KUKA KRL program: ConfGarra.src, ConfGarra.dat

--- ConfGarra.src ---
&ACCESS RVO1
&PARAM EDITMASK = *
DEF ConfGarra( )

      SWITCH ConfGarraOp
         CASE 11
            Abre_Gar_Triplo_Lado_A = TRUE
            Fecha_Gar_Triplo_Lado_A = FALSE

            Abre_Gar_Triplo_Lado_B = FALSE
            Fecha_Gar_Triplo_Lado_B = TRUE

            Abre_Comp_Indiv_Gar_1 = FALSE
            Fecha_Comp_Indiv_Gar_1 = TRUE

            Abre_Comp_Indiv_Gar_3 = TRUE
            Fecha_Comp_Indiv_Gar_3 = FALSE

            Abre_Comp_Indiv_Gar_4 = FALSE
            Fecha_Comp_Indiv_Gar_4 = TRUE

            Abre_Comp_Indiv_Gar_6 = TRUE
            Fecha_Comp_Indiv_Gar_6 = FALSE

            Ava_Cil_2_Gar_1 = TRUE
            Rec_Cil_2_Gar_1 = FALSE

            Ava_Cil_2_Gar_2 = TRUE
            Rec_Cil_2_Gar_2 = FALSE

            Ava_Cil_2_Gar_3 = TRUE
            Rec_Cil_2_Gar_3 = FALSE

            Ava_Cil_2_Gar_4 = TRUE
            Rec_Cil_2_Gar_4 = FALSE

            Ava_Cil_2_Gar_5 = TRUE
            Rec_Cil_2_Gar_5 = FALSE

            Ava_Cil_2_Gar_6 = TRUE
            Rec_Cil_2_Gar_6 = FALSE

            Ava_Cil_1_Gar_1 = TRUE
            Rec_Cil_1_Gar_1 = FALSE

            Ava_Cil_1_Gar_2 = TRUE
            Rec_Cil_1_Gar_2 = FALSE

            Ava_Cil_1_Gar_3 = TRUE
            Rec_Cil_1_Gar_3 = FALSE

            Ava_Cil_1_Gar_4 = TRUE
            Rec_Cil_1_Gar_4 = FALSE

            Ava_Cil_1_Gar_5 = TRUE
            Rec_Cil_1_Gar_5 = FALSE

            Ava_Cil_1_Gar_6 = TRUE
            Rec_Cil_1_Gar_6 = FALSE

            WAIT FOR ( Cil_Comp_Triplo_A_Ava == FALSE )
            WAIT FOR ( Cil_Comp_Triplo_A_Rec == TRUE )
            WAIT FOR ( Cil_Comp_Triplo_B_Ava == TRUE )
            WAIT FOR ( Cil_Comp_Triplo_B_Rec == FALSE )
            WAIT FOR ( Cil_Comp_Indiv_Gr_1_Aber == FALSE )
            WAIT FOR ( Cil_Comp_Indiv_Gr_1_Fech == TRUE )
            WAIT FOR ( Cil_Comp_Indiv_Gr_3_Aber == TRUE )
            WAIT FOR ( Cil_Comp_Indiv_Gr_3_Fech == FALSE )
            WAIT FOR ( Cil_Comp_Indiv_Gr_4_Aber == FALSE )
            WAIT FOR ( Cil_Comp_Indiv_Gr_4_Fech == TRUE )
            WAIT FOR ( Cil_Comp_Indiv_Gr_6_Aber == TRUE )
            WAIT FOR ( Cil_Comp_Indiv_Gr_6_Fech == FALSE )
            WAIT FOR ( Cil_2_Gar_1_Ava == TRUE )
            WAIT FOR ( Cil_2_Gar_2_Ava == TRUE )
            WAIT FOR ( Cil_2_Gar_3_Ava == TRUE )
            WAIT FOR ( Cil_2_Gar_4_Ava == TRUE )
            WAIT FOR ( Cil_2_Gar_5_Ava == TRUE )
            WAIT FOR ( Cil_2_Gar_6_Ava == TRUE )
            WAIT FOR ( Cil_1_Gar_1_Ava == TRUE )
            WAIT FOR ( Cil_1_Gar_2_Ava == TRUE )
            WAIT FOR ( Cil_1_Gar_3_Ava == TRUE )
            WAIT FOR ( Cil_1_Gar_4_Ava == TRUE )
            WAIT FOR ( Cil_1_Gar_5_Ava == TRUE )
            WAIT FOR ( Cil_1_Gar_6_Ava == TRUE )

         CASE 21
            Abre_Gar_Triplo_Lado_A = FALSE
            Fecha_Gar_Triplo_Lado_A = TRUE

            Abre_Gar_Triplo_Lado_B = FALSE
            Fecha_Gar_Triplo_Lado_B = TRUE

            Abre_Comp_Indiv_Gar_1 = FALSE
            Fecha_Comp_Indiv_Gar_1 = TRUE

            Abre_Comp_Indiv_Gar_3 = FALSE
            Fecha_Comp_Indiv_Gar_3 = TRUE

            Abre_Comp_Indiv_Gar_4 = FALSE
            Fecha_Comp_Indiv_Gar_4 = TRUE

            Abre_Comp_Indiv_Gar_6 = FALSE
            Fecha_Comp_Indiv_Gar_6 = TRUE

            Ava_Cil_2_Gar_1 = TRUE
            Rec_Cil_2_Gar_1 = FALSE

            Ava_Cil_2_Gar_2 = TRUE
            Rec_Cil_2_Gar_2 = FALSE

            Ava_Cil_2_Gar_3 = TRUE
            Rec_Cil_2_Gar_3 = FALSE

            Ava_Cil_2_Gar_4 = TRUE
            Rec_Cil_2_Gar_4 = FALSE

            Ava_Cil_2_Gar_5 = TRUE
            Rec_Cil_2_Gar_5 = FALSE

            Ava_Cil_2_Gar_6 = TRUE
            Rec_Cil_2_Gar_6 = FALSE

            Ava_Cil_1_Gar_1 = TRUE
            Rec_Cil_1_Gar_1 = FALSE

            Ava_Cil_1_Gar_2 = TRUE
            Rec_Cil_1_Gar_2 = FALSE

            Ava_Cil_1_Gar_3 = TRUE
            Rec_Cil_1_Gar_3 = FALSE

            Ava_Cil_1_Gar_4 = TRUE
            Rec_Cil_1_Gar_4 = FALSE

            Ava_Cil_1_Gar_5 = TRUE
            Rec_Cil_1_Gar_5 = FALSE

            Ava_Cil_1_Gar_6 = TRUE
            Rec_Cil_1_Gar_6 = FALSE

            WAIT FOR ( Cil_Comp_Triplo_A_Ava == TRUE )
            WAIT FOR ( Cil_Comp_Triplo_A_Rec == FALSE )
            WAIT FOR ( Cil_Comp_Triplo_B_Ava == TRUE )
            WAIT FOR ( Cil_Comp_Triplo_B_Rec == FALSE )
            WAIT FOR ( Cil_Comp_Indiv_Gr_1_Aber == FALSE )
            WAIT FOR ( Cil_Comp_Indiv_Gr_1_Fech == TRUE )
            WAIT FOR ( Cil_Comp_Indiv_Gr_3_Aber == FALSE )
            WAIT FOR ( Cil_Comp_Indiv_Gr_3_Fech == TRUE )
            WAIT FOR ( Cil_Comp_Indiv_Gr_4_Aber == FALSE )
            WAIT FOR ( Cil_Comp_Indiv_Gr_4_Fech == TRUE )
            WAIT FOR ( Cil_Comp_Indiv_Gr_6_Aber == FALSE )
            WAIT FOR ( Cil_Comp_Indiv_Gr_6_Fech == TRUE )
            WAIT FOR ( Cil_2_Gar_1_Ava == TRUE )
            WAIT FOR ( Cil_2_Gar_2_Ava == TRUE )
            WAIT FOR ( Cil_2_Gar_3_Ava == TRUE )
            WAIT FOR ( Cil_2_Gar_4_Ava == TRUE )
            WAIT FOR ( Cil_2_Gar_5_Ava == TRUE )
            WAIT FOR ( Cil_2_Gar_6_Ava == TRUE )
            WAIT FOR ( Cil_1_Gar_1_Ava == TRUE )
            WAIT FOR ( Cil_1_Gar_2_Ava == TRUE )
            WAIT FOR ( Cil_1_Gar_3_Ava == TRUE )
            WAIT FOR ( Cil_1_Gar_4_Ava == TRUE )
            WAIT FOR ( Cil_1_Gar_5_Ava == TRUE )
            WAIT FOR ( Cil_1_Gar_6_Ava == TRUE )

         CASE 101
            Abre_Gar_Triplo_Lado_A = TRUE
            Fecha_Gar_Triplo_Lado_A = FALSE

            Abre_Gar_Triplo_Lado_B = TRUE
            Fecha_Gar_Triplo_Lado_B = FALSE

            Abre_Comp_Indiv_Gar_1 = TRUE
            Fecha_Comp_Indiv_Gar_1 = FALSE

            Abre_Comp_Indiv_Gar_3 = FALSE
            Fecha_Comp_Indiv_Gar_3 = TRUE

            Abre_Comp_Indiv_Gar_4 = FALSE
            Fecha_Comp_Indiv_Gar_4 = TRUE

            Abre_Comp_Indiv_Gar_6 = TRUE
            Fecha_Comp_Indiv_Gar_6 = FALSE

            Ava_Cil_2_Gar_1 = TRUE
            Rec_Cil_2_Gar_1 = FALSE

            Ava_Cil_2_Gar_2 = TRUE
            Rec_Cil_2_Gar_2 = FALSE

            Ava_Cil_2_Gar_3 = TRUE
            Rec_Cil_2_Gar_3 = FALSE

            Ava_Cil_2_Gar_4 = TRUE
            Rec_Cil_2_Gar_4 = FALSE

            Ava_Cil_2_Gar_5 = TRUE
            Rec_Cil_2_Gar_5 = FALSE

            Ava_Cil_2_Gar_6 = TRUE
            Rec_Cil_2_Gar_6 = FALSE

            Ava_Cil_1_Gar_1 = TRUE
            Rec_Cil_1_Gar_1 = FALSE

            Ava_Cil_1_Gar_2 = TRUE
            Rec_Cil_1_Gar_2 = FALSE

            Ava_Cil_1_Gar_3 = TRUE
            Rec_Cil_1_Gar_3 = FALSE

            Ava_Cil_1_Gar_4 = TRUE
            Rec_Cil_1_Gar_4 = FALSE

            Ava_Cil_1_Gar_5 = TRUE
            Rec_Cil_1_Gar_5 = FALSE

            Ava_Cil_1_Gar_6 = TRUE
            Rec_Cil_1_Gar_6 = FALSE

            WAIT FOR ( Cil_Comp_Triplo_A_Ava == FALSE )
            WAIT FOR ( Cil_Comp_Triplo_A_Rec == TRUE )
            WAIT FOR ( Cil_Comp_Triplo_B_Ava == FALSE )
            WAIT FOR ( Cil_Comp_Triplo_B_Rec == TRUE )
            WAIT FOR ( Cil_Comp_Indiv_Gr_1_Aber == TRUE )
            WAIT FOR ( Cil_Comp_Indiv_Gr_1_Fech == FALSE )
            WAIT FOR ( Cil_Comp_Indiv_Gr_3_Aber == FALSE )
            WAIT FOR ( Cil_Comp_Indiv_Gr_3_Fech == TRUE )
            WAIT FOR ( Cil_Comp_Indiv_Gr_4_Aber == FALSE )
            WAIT FOR ( Cil_Comp_Indiv_Gr_4_Fech == TRUE )
            WAIT FOR ( Cil_Comp_Indiv_Gr_6_Aber == TRUE )
            WAIT FOR ( Cil_Comp_Indiv_Gr_6_Fech == FALSE )
            WAIT FOR ( Cil_2_Gar_1_Ava == TRUE )
            WAIT FOR ( Cil_2_Gar_2_Ava == TRUE )
            WAIT FOR ( Cil_2_Gar_3_Ava == TRUE )
            WAIT FOR ( Cil_2_Gar_4_Ava == TRUE )
            WAIT FOR ( Cil_2_Gar_5_Ava == TRUE )
            WAIT FOR ( Cil_2_Gar_6_Ava == TRUE )
            WAIT FOR ( Cil_1_Gar_1_Ava == TRUE )
            WAIT FOR ( Cil_1_Gar_2_Ava == TRUE )
            WAIT FOR ( Cil_1_Gar_3_Ava == TRUE )
            WAIT FOR ( Cil_1_Gar_4_Ava == TRUE )
            WAIT FOR ( Cil_1_Gar_5_Ava == TRUE )
            WAIT FOR ( Cil_1_Gar_6_Ava == TRUE )

         CASE 102
            Abre_Gar_Triplo_Lado_A = TRUE
            Fecha_Gar_Triplo_Lado_A = FALSE

            Abre_Gar_Triplo_Lado_B = TRUE
            Fecha_Gar_Triplo_Lado_B = FALSE

            Abre_Comp_Indiv_Gar_1 = TRUE
            Fecha_Comp_Indiv_Gar_1 = FALSE

            Abre_Comp_Indiv_Gar_3 = FALSE
            Fecha_Comp_Indiv_Gar_3 = TRUE

            Abre_Comp_Indiv_Gar_4 = FALSE
            Fecha_Comp_Indiv_Gar_4 = TRUE

            Abre_Comp_Indiv_Gar_6 = TRUE
            Fecha_Comp_Indiv_Gar_6 = FALSE

            Ava_Cil_1_Gar_1 = TRUE
            Rec_Cil_1_Gar_1 = FALSE

            Ava_Cil_1_Gar_2 = TRUE
            Rec_Cil_1_Gar_2 = FALSE

            Ava_Cil_1_Gar_3 = TRUE
            Rec_Cil_1_Gar_3 = FALSE

            Ava_Cil_1_Gar_4 = TRUE
            Rec_Cil_1_Gar_4 = FALSE

            Ava_Cil_1_Gar_5 = TRUE
            Rec_Cil_1_Gar_5 = FALSE

            Ava_Cil_1_Gar_6 = TRUE
            Rec_Cil_1_Gar_6 = FALSE

            Ava_Cil_2_Gar_1 = TRUE
            Rec_Cil_2_Gar_1 = FALSE

            Ava_Cil_2_Gar_2 = TRUE
            Rec_Cil_2_Gar_2 = FALSE

            Ava_Cil_2_Gar_3 = TRUE
            Rec_Cil_2_Gar_3 = FALSE

            Ava_Cil_2_Gar_4 = TRUE
            Rec_Cil_2_Gar_4 = FALSE

            Ava_Cil_2_Gar_5 = TRUE
            Rec_Cil_2_Gar_5 = FALSE

            Ava_Cil_2_Gar_6 = TRUE
            Rec_Cil_2_Gar_6 = FALSE

            WAIT FOR ( Cil_Comp_Triplo_A_Ava == FALSE )
            WAIT FOR ( Cil_Comp_Triplo_A_Rec == TRUE )
            WAIT FOR ( Cil_Comp_Triplo_B_Ava == FALSE )
            WAIT FOR ( Cil_Comp_Triplo_B_Rec == TRUE )
            WAIT FOR ( Cil_Comp_Indiv_Gr_1_Aber == TRUE )
            WAIT FOR ( Cil_Comp_Indiv_Gr_1_Fech == FALSE )
            WAIT FOR ( Cil_Comp_Indiv_Gr_3_Aber == FALSE )
            WAIT FOR ( Cil_Comp_Indiv_Gr_3_Fech == TRUE )
            WAIT FOR ( Cil_Comp_Indiv_Gr_4_Aber == FALSE )
            WAIT FOR ( Cil_Comp_Indiv_Gr_4_Fech == TRUE )
            WAIT FOR ( Cil_Comp_Indiv_Gr_6_Aber == TRUE )
            WAIT FOR ( Cil_Comp_Indiv_Gr_6_Fech == FALSE )
            WAIT FOR ( Cil_1_Gar_1_Ava == TRUE )
            WAIT FOR ( Cil_1_Gar_2_Ava == TRUE )
            WAIT FOR ( Cil_1_Gar_3_Ava == TRUE )
            WAIT FOR ( Cil_1_Gar_4_Ava == TRUE )
            WAIT FOR ( Cil_1_Gar_5_Ava == TRUE )
            WAIT FOR ( Cil_1_Gar_6_Ava == TRUE )
            WAIT FOR ( Cil_2_Gar_1_Ava == TRUE )
            WAIT FOR ( Cil_2_Gar_2_Ava == TRUE )
            WAIT FOR ( Cil_2_Gar_3_Ava == TRUE )
            WAIT FOR ( Cil_2_Gar_4_Ava == TRUE )
            WAIT FOR ( Cil_2_Gar_5_Ava == TRUE )
            WAIT FOR ( Cil_2_Gar_6_Ava == TRUE )

         CASE 121
            Abre_Gar_Triplo_Lado_A = TRUE
            Fecha_Gar_Triplo_Lado_A = FALSE

            Abre_Gar_Triplo_Lado_B = TRUE
            Fecha_Gar_Triplo_Lado_B = FALSE

            Abre_Comp_Indiv_Gar_1 = FALSE
            Fecha_Comp_Indiv_Gar_1 = TRUE

            Abre_Comp_Indiv_Gar_3 = FALSE
            Fecha_Comp_Indiv_Gar_3 = TRUE

            Abre_Comp_Indiv_Gar_4 = FALSE
            Fecha_Comp_Indiv_Gar_4 = TRUE

            Abre_Comp_Indiv_Gar_6 = FALSE
            Fecha_Comp_Indiv_Gar_6 = TRUE

            Ava_Cil_1_Gar_1 = TRUE
            Rec_Cil_1_Gar_1 = FALSE

            Ava_Cil_1_Gar_2 = TRUE
            Rec_Cil_1_Gar_2 = FALSE

            Ava_Cil_1_Gar_3 = TRUE
            Rec_Cil_1_Gar_3 = FALSE

            Ava_Cil_1_Gar_4 = TRUE
            Rec_Cil_1_Gar_4 = FALSE

            Ava_Cil_1_Gar_5 = TRUE
            Rec_Cil_1_Gar_5 = FALSE

            Ava_Cil_1_Gar_6 = TRUE
            Rec_Cil_1_Gar_6 = FALSE

            Ava_Cil_2_Gar_1 = TRUE
            Rec_Cil_2_Gar_1 = FALSE

            Ava_Cil_2_Gar_2 = TRUE
            Rec_Cil_2_Gar_2 = FALSE

            Ava_Cil_2_Gar_3 = TRUE
            Rec_Cil_2_Gar_3 = FALSE

            Ava_Cil_2_Gar_4 = TRUE
            Rec_Cil_2_Gar_4 = FALSE

            Ava_Cil_2_Gar_5 = TRUE
            Rec_Cil_2_Gar_5 = FALSE

            Ava_Cil_2_Gar_6 = TRUE
            Rec_Cil_2_Gar_6 = FALSE

            WAIT FOR ( Cil_Comp_Triplo_A_Ava == TRUE )
            WAIT FOR ( Cil_Comp_Triplo_A_Rec == FALSE )
            WAIT FOR ( Cil_Comp_Triplo_B_Ava == TRUE )
            WAIT FOR ( Cil_Comp_Triplo_B_Rec == FALSE )
            WAIT FOR ( Cil_Comp_Indiv_Gr_1_Aber == FALSE )
            WAIT FOR ( Cil_Comp_Indiv_Gr_1_Fech == TRUE )
            WAIT FOR ( Cil_Comp_Indiv_Gr_3_Aber == FALSE )
            WAIT FOR ( Cil_Comp_Indiv_Gr_3_Fech == TRUE )
            WAIT FOR ( Cil_Comp_Indiv_Gr_4_Aber == FALSE )
            WAIT FOR ( Cil_Comp_Indiv_Gr_4_Fech == TRUE )
            WAIT FOR ( Cil_Comp_Indiv_Gr_6_Aber == FALSE )
            WAIT FOR ( Cil_Comp_Indiv_Gr_6_Fech == TRUE )
            WAIT FOR ( Cil_1_Gar_1_Ava == TRUE )
            WAIT FOR ( Cil_1_Gar_2_Ava == TRUE )
            WAIT FOR ( Cil_1_Gar_3_Ava == TRUE )
            WAIT FOR ( Cil_1_Gar_4_Ava == TRUE )
            WAIT FOR ( Cil_1_Gar_5_Ava == TRUE )
            WAIT FOR ( Cil_1_Gar_6_Ava == TRUE )
            WAIT FOR ( Cil_2_Gar_1_Ava == TRUE )
            WAIT FOR ( Cil_2_Gar_2_Ava == TRUE )
            WAIT FOR ( Cil_2_Gar_3_Ava == TRUE )
            WAIT FOR ( Cil_2_Gar_4_Ava == TRUE )
            WAIT FOR ( Cil_2_Gar_5_Ava == TRUE )
            WAIT FOR ( Cil_2_Gar_6_Ava == TRUE )

         CASE 122
            Abre_Gar_Triplo_Lado_A = TRUE
            Fecha_Gar_Triplo_Lado_A = FALSE

            Abre_Gar_Triplo_Lado_B = TRUE
            Fecha_Gar_Triplo_Lado_B = FALSE

            Abre_Comp_Indiv_Gar_1 = TRUE
            Fecha_Comp_Indiv_Gar_1 = FALSE

            Abre_Comp_Indiv_Gar_3 = FALSE
            Fecha_Comp_Indiv_Gar_3 = TRUE

            Abre_Comp_Indiv_Gar_4 = FALSE
            Fecha_Comp_Indiv_Gar_4 = TRUE

            Abre_Comp_Indiv_Gar_6 = TRUE
            Fecha_Comp_Indiv_Gar_6 = FALSE

            Ava_Cil_1_Gar_1 = TRUE
            Rec_Cil_1_Gar_1 = FALSE

            Ava_Cil_1_Gar_2 = TRUE
            Rec_Cil_1_Gar_2 = FALSE

            Ava_Cil_1_Gar_3 = TRUE
            Rec_Cil_1_Gar_3 = FALSE

            Ava_Cil_1_Gar_4 = TRUE
            Rec_Cil_1_Gar_4 = FALSE

            Ava_Cil_1_Gar_5 = TRUE
            Rec_Cil_1_Gar_5 = FALSE

            Ava_Cil_1_Gar_6 = TRUE
            Rec_Cil_1_Gar_6 = FALSE

            Ava_Cil_2_Gar_1 = TRUE
            Rec_Cil_2_Gar_1 = FALSE

            Ava_Cil_2_Gar_2 = TRUE
            Rec_Cil_2_Gar_2 = FALSE

            Ava_Cil_2_Gar_3 = TRUE
            Rec_Cil_2_Gar_3 = FALSE

            Ava_Cil_2_Gar_4 = TRUE
            Rec_Cil_2_Gar_4 = FALSE

            Ava_Cil_2_Gar_5 = TRUE
            Rec_Cil_2_Gar_5 = FALSE

            Ava_Cil_2_Gar_6 = TRUE
            Rec_Cil_2_Gar_6 = FALSE

            WAIT FOR ( Cil_Comp_Triplo_A_Ava == TRUE )
            WAIT FOR ( Cil_Comp_Triplo_A_Rec == FALSE )
            WAIT FOR ( Cil_Comp_Triplo_B_Ava == TRUE )
            WAIT FOR ( Cil_Comp_Triplo_B_Rec == FALSE )
            WAIT FOR ( Cil_Comp_Indiv_Gr_1_Aber == TRUE )
            WAIT FOR ( Cil_Comp_Indiv_Gr_1_Fech == FALSE )
            WAIT FOR ( Cil_Comp_Indiv_Gr_3_Aber == FALSE )
            WAIT FOR ( Cil_Comp_Indiv_Gr_3_Fech == TRUE )
            WAIT FOR ( Cil_Comp_Indiv_Gr_4_Aber == FALSE )
            WAIT FOR ( Cil_Comp_Indiv_Gr_4_Fech == TRUE )
            WAIT FOR ( Cil_Comp_Indiv_Gr_6_Aber == TRUE )
            WAIT FOR ( Cil_Comp_Indiv_Gr_6_Fech == FALSE )
            WAIT FOR ( Cil_1_Gar_1_Ava == TRUE )
            WAIT FOR ( Cil_1_Gar_2_Ava == TRUE )
            WAIT FOR ( Cil_1_Gar_3_Ava == TRUE )
            WAIT FOR ( Cil_1_Gar_4_Ava == TRUE )
            WAIT FOR ( Cil_1_Gar_5_Ava == TRUE )
            WAIT FOR ( Cil_1_Gar_6_Ava == TRUE )
            WAIT FOR ( Cil_2_Gar_1_Ava == TRUE )
            WAIT FOR ( Cil_2_Gar_2_Ava == TRUE )
            WAIT FOR ( Cil_2_Gar_3_Ava == TRUE )
            WAIT FOR ( Cil_2_Gar_4_Ava == TRUE )
            WAIT FOR ( Cil_2_Gar_5_Ava == TRUE )
            WAIT FOR ( Cil_2_Gar_6_Ava == TRUE )

         CASE 31
            Abre_Gar_Triplo_Lado_A = TRUE
            Fecha_Gar_Triplo_Lado_A = FALSE

            Abre_Gar_Triplo_Lado_B = TRUE
            Fecha_Gar_Triplo_Lado_B = FALSE

            Abre_Comp_Indiv_Gar_1 = FALSE
            Fecha_Comp_Indiv_Gar_1 = TRUE

            Abre_Comp_Indiv_Gar_3 = FALSE
            Fecha_Comp_Indiv_Gar_3 = TRUE

            Abre_Comp_Indiv_Gar_4 = FALSE
            Fecha_Comp_Indiv_Gar_4 = TRUE

            Abre_Comp_Indiv_Gar_6 = FALSE
            Fecha_Comp_Indiv_Gar_6 = TRUE

            Ava_Cil_1_Gar_1 = TRUE
            Rec_Cil_1_Gar_1 = FALSE

            Ava_Cil_1_Gar_2 = TRUE
            Rec_Cil_1_Gar_2 = FALSE

            Ava_Cil_1_Gar_3 = TRUE
            Rec_Cil_1_Gar_3 = FALSE

            Ava_Cil_1_Gar_4 = TRUE
            Rec_Cil_1_Gar_4 = FALSE

            Ava_Cil_1_Gar_5 = TRUE
            Rec_Cil_1_Gar_5 = FALSE

            Ava_Cil_1_Gar_6 = TRUE
            Rec_Cil_1_Gar_6 = FALSE

            Ava_Cil_2_Gar_1 = TRUE
            Rec_Cil_2_Gar_1 = FALSE

            Ava_Cil_2_Gar_2 = TRUE
            Rec_Cil_2_Gar_2 = FALSE

            Ava_Cil_2_Gar_3 = TRUE
            Rec_Cil_2_Gar_3 = FALSE

            Ava_Cil_2_Gar_4 = TRUE
            Rec_Cil_2_Gar_4 = FALSE

            Ava_Cil_2_Gar_5 = TRUE
            Rec_Cil_2_Gar_5 = FALSE

            Ava_Cil_2_Gar_6 = TRUE
            Rec_Cil_2_Gar_6 = FALSE

            WAIT FOR ( Cil_Comp_Triplo_A_Ava == TRUE )
            WAIT FOR ( Cil_Comp_Triplo_A_Rec == FALSE )
            WAIT FOR ( Cil_Comp_Triplo_B_Ava == TRUE )
            WAIT FOR ( Cil_Comp_Triplo_B_Rec == FALSE )
            WAIT FOR ( Cil_Comp_Indiv_Gr_1_Aber == FALSE )
            WAIT FOR ( Cil_Comp_Indiv_Gr_1_Fech == TRUE )
            WAIT FOR ( Cil_Comp_Indiv_Gr_3_Aber == FALSE )
            WAIT FOR ( Cil_Comp_Indiv_Gr_3_Fech == TRUE )
            WAIT FOR ( Cil_Comp_Indiv_Gr_4_Aber == FALSE )
            WAIT FOR ( Cil_Comp_Indiv_Gr_4_Fech == TRUE )
            WAIT FOR ( Cil_Comp_Indiv_Gr_6_Aber == FALSE )
            WAIT FOR ( Cil_Comp_Indiv_Gr_6_Fech == TRUE )
            WAIT FOR ( Cil_1_Gar_1_Ava == TRUE )
            WAIT FOR ( Cil_1_Gar_2_Ava == TRUE )
            WAIT FOR ( Cil_1_Gar_3_Ava == TRUE )
            WAIT FOR ( Cil_1_Gar_4_Ava == TRUE )
            WAIT FOR ( Cil_1_Gar_5_Ava == TRUE )
            WAIT FOR ( Cil_1_Gar_6_Ava == TRUE )
            WAIT FOR ( Cil_2_Gar_1_Ava == TRUE )
            WAIT FOR ( Cil_2_Gar_2_Ava == TRUE )
            WAIT FOR ( Cil_2_Gar_3_Ava == TRUE )
            WAIT FOR ( Cil_2_Gar_4_Ava == TRUE )
            WAIT FOR ( Cil_2_Gar_5_Ava == TRUE )
            WAIT FOR ( Cil_2_Gar_6_Ava == TRUE )

         CASE 32
            Abre_Gar_Triplo_Lado_A = TRUE
            Fecha_Gar_Triplo_Lado_A = FALSE

            Abre_Gar_Triplo_Lado_B = TRUE
            Fecha_Gar_Triplo_Lado_B = FALSE

            Abre_Comp_Indiv_Gar_1 = FALSE
            Fecha_Comp_Indiv_Gar_1 = TRUE

            Abre_Comp_Indiv_Gar_3 = FALSE
            Fecha_Comp_Indiv_Gar_3 = TRUE

            Abre_Comp_Indiv_Gar_4 = FALSE
            Fecha_Comp_Indiv_Gar_4 = TRUE

            Abre_Comp_Indiv_Gar_6 = FALSE
            Fecha_Comp_Indiv_Gar_6 = TRUE

            Ava_Cil_1_Gar_1 = TRUE
            Rec_Cil_1_Gar_1 = FALSE

            Ava_Cil_1_Gar_2 = TRUE
            Rec_Cil_1_Gar_2 = FALSE

            Ava_Cil_1_Gar_3 = TRUE
            Rec_Cil_1_Gar_3 = FALSE

            Ava_Cil_1_Gar_4 = TRUE
            Rec_Cil_1_Gar_4 = FALSE

            Ava_Cil_1_Gar_5 = TRUE
            Rec_Cil_1_Gar_5 = FALSE

            Ava_Cil_1_Gar_6 = TRUE
            Rec_Cil_1_Gar_6 = FALSE

            Ava_Cil_2_Gar_1 = TRUE
            Rec_Cil_2_Gar_1 = FALSE

            Ava_Cil_2_Gar_2 = TRUE
            Rec_Cil_2_Gar_2 = FALSE

            Ava_Cil_2_Gar_3 = TRUE
            Rec_Cil_2_Gar_3 = FALSE

            Ava_Cil_2_Gar_4 = TRUE
            Rec_Cil_2_Gar_4 = FALSE

            Ava_Cil_2_Gar_5 = TRUE
            Rec_Cil_2_Gar_5 = FALSE

            Ava_Cil_2_Gar_6 = TRUE
            Rec_Cil_2_Gar_6 = FALSE

            WAIT FOR ( Cil_Comp_Triplo_A_Ava == TRUE )
            WAIT FOR ( Cil_Comp_Triplo_A_Rec == FALSE )
            WAIT FOR ( Cil_Comp_Triplo_B_Ava == TRUE )
            WAIT FOR ( Cil_Comp_Triplo_B_Rec == FALSE )
            WAIT FOR ( Cil_Comp_Indiv_Gr_1_Aber == FALSE )
            WAIT FOR ( Cil_Comp_Indiv_Gr_1_Fech == TRUE )
            WAIT FOR ( Cil_Comp_Indiv_Gr_3_Aber == FALSE )
            WAIT FOR ( Cil_Comp_Indiv_Gr_3_Fech == TRUE )
            WAIT FOR ( Cil_Comp_Indiv_Gr_4_Aber == FALSE )
            WAIT FOR ( Cil_Comp_Indiv_Gr_4_Fech == TRUE )
            WAIT FOR ( Cil_Comp_Indiv_Gr_6_Aber == FALSE )
            WAIT FOR ( Cil_Comp_Indiv_Gr_6_Fech == TRUE )
            WAIT FOR ( Cil_1_Gar_1_Ava == TRUE )
            WAIT FOR ( Cil_1_Gar_2_Ava == TRUE )
            WAIT FOR ( Cil_1_Gar_3_Ava == TRUE )
            WAIT FOR ( Cil_1_Gar_4_Ava == TRUE )
            WAIT FOR ( Cil_1_Gar_5_Ava == TRUE )
            WAIT FOR ( Cil_1_Gar_6_Ava == TRUE )
            WAIT FOR ( Cil_2_Gar_1_Ava == TRUE )
            WAIT FOR ( Cil_2_Gar_2_Ava == TRUE )
            WAIT FOR ( Cil_2_Gar_3_Ava == TRUE )
            WAIT FOR ( Cil_2_Gar_4_Ava == TRUE )
            WAIT FOR ( Cil_2_Gar_5_Ava == TRUE )
            WAIT FOR ( Cil_2_Gar_6_Ava == TRUE )

         CASE 111
            Abre_Gar_Triplo_Lado_A = TRUE
            Fecha_Gar_Triplo_Lado_A = FALSE

            Abre_Gar_Triplo_Lado_B = TRUE
            Fecha_Gar_Triplo_Lado_B = FALSE

            Abre_Comp_Indiv_Gar_1 = FALSE
            Fecha_Comp_Indiv_Gar_1 = TRUE

            Abre_Comp_Indiv_Gar_3 = FALSE
            Fecha_Comp_Indiv_Gar_3 = TRUE

            Abre_Comp_Indiv_Gar_4 = FALSE
            Fecha_Comp_Indiv_Gar_4 = TRUE

            Abre_Comp_Indiv_Gar_6 = FALSE
            Fecha_Comp_Indiv_Gar_6 = TRUE

            Ava_Cil_1_Gar_1 = TRUE
            Rec_Cil_1_Gar_1 = FALSE

            Ava_Cil_1_Gar_2 = TRUE
            Rec_Cil_1_Gar_2 = FALSE

            Ava_Cil_1_Gar_3 = TRUE
            Rec_Cil_1_Gar_3 = FALSE

            Ava_Cil_1_Gar_4 = TRUE
            Rec_Cil_1_Gar_4 = FALSE

            Ava_Cil_1_Gar_5 = TRUE
            Rec_Cil_1_Gar_5 = FALSE

            Ava_Cil_1_Gar_6 = TRUE
            Rec_Cil_1_Gar_6 = FALSE

            Ava_Cil_2_Gar_1 = TRUE
            Rec_Cil_2_Gar_1 = FALSE

            Ava_Cil_2_Gar_2 = TRUE
            Rec_Cil_2_Gar_2 = FALSE

            Ava_Cil_2_Gar_3 = TRUE
            Rec_Cil_2_Gar_3 = FALSE

            Ava_Cil_2_Gar_4 = TRUE
            Rec_Cil_2_Gar_4 = FALSE

            Ava_Cil_2_Gar_5 = TRUE
            Rec_Cil_2_Gar_5 = FALSE

            Ava_Cil_2_Gar_6 = TRUE
            Rec_Cil_2_Gar_6 = FALSE

            WAIT FOR ( Cil_Comp_Triplo_A_Ava == TRUE )
            WAIT FOR ( Cil_Comp_Triplo_A_Rec == FALSE )
            WAIT FOR ( Cil_Comp_Triplo_B_Ava == TRUE )
            WAIT FOR ( Cil_Comp_Triplo_B_Rec == FALSE )
            WAIT FOR ( Cil_Comp_Indiv_Gr_1_Aber == FALSE )
            WAIT FOR ( Cil_Comp_Indiv_Gr_1_Fech == TRUE )
            WAIT FOR ( Cil_Comp_Indiv_Gr_3_Aber == FALSE )
            WAIT FOR ( Cil_Comp_Indiv_Gr_3_Fech == TRUE )
            WAIT FOR ( Cil_Comp_Indiv_Gr_4_Aber == FALSE )
            WAIT FOR ( Cil_Comp_Indiv_Gr_4_Fech == TRUE )
            WAIT FOR ( Cil_Comp_Indiv_Gr_6_Aber == FALSE )
            WAIT FOR ( Cil_Comp_Indiv_Gr_6_Fech == TRUE )
            WAIT FOR ( Cil_1_Gar_1_Ava == TRUE )
            WAIT FOR ( Cil_1_Gar_2_Ava == TRUE )
            WAIT FOR ( Cil_1_Gar_3_Ava == TRUE )
            WAIT FOR ( Cil_1_Gar_4_Ava == TRUE )
            WAIT FOR ( Cil_1_Gar_5_Ava == TRUE )
            WAIT FOR ( Cil_1_Gar_6_Ava == TRUE )
            WAIT FOR ( Cil_2_Gar_1_Ava == TRUE )
            WAIT FOR ( Cil_2_Gar_2_Ava == TRUE )
            WAIT FOR ( Cil_2_Gar_3_Ava == TRUE )
            WAIT FOR ( Cil_2_Gar_4_Ava == TRUE )
            WAIT FOR ( Cil_2_Gar_5_Ava == TRUE )
            WAIT FOR ( Cil_2_Gar_6_Ava == TRUE )

         CASE 112
            Abre_Gar_Triplo_Lado_A = TRUE
            Fecha_Gar_Triplo_Lado_A = FALSE

            Abre_Gar_Triplo_Lado_B = TRUE
            Fecha_Gar_Triplo_Lado_B = FALSE

            Abre_Comp_Indiv_Gar_1 = FALSE
            Fecha_Comp_Indiv_Gar_1 = TRUE

            Abre_Comp_Indiv_Gar_3 = FALSE
            Fecha_Comp_Indiv_Gar_3 = TRUE

            Abre_Comp_Indiv_Gar_4 = FALSE
            Fecha_Comp_Indiv_Gar_4 = TRUE

            Abre_Comp_Indiv_Gar_6 = FALSE
            Fecha_Comp_Indiv_Gar_6 = TRUE

            Ava_Cil_1_Gar_1 = TRUE
            Rec_Cil_1_Gar_1 = FALSE

            Ava_Cil_1_Gar_2 = TRUE
            Rec_Cil_1_Gar_2 = FALSE

            Ava_Cil_1_Gar_3 = TRUE
            Rec_Cil_1_Gar_3 = FALSE

            Ava_Cil_1_Gar_4 = TRUE
            Rec_Cil_1_Gar_4 = FALSE

            Ava_Cil_1_Gar_5 = TRUE
            Rec_Cil_1_Gar_5 = FALSE

            Ava_Cil_1_Gar_6 = TRUE
            Rec_Cil_1_Gar_6 = FALSE

            Ava_Cil_2_Gar_1 = TRUE
            Rec_Cil_2_Gar_1 = FALSE

            Ava_Cil_2_Gar_2 = TRUE
            Rec_Cil_2_Gar_2 = FALSE

            Ava_Cil_2_Gar_3 = TRUE
            Rec_Cil_2_Gar_3 = FALSE

            Ava_Cil_2_Gar_4 = TRUE
            Rec_Cil_2_Gar_4 = FALSE

            Ava_Cil_2_Gar_5 = TRUE
            Rec_Cil_2_Gar_5 = FALSE

            Ava_Cil_2_Gar_6 = TRUE
            Rec_Cil_2_Gar_6 = FALSE

            WAIT FOR ( Cil_Comp_Triplo_A_Ava == TRUE )
            WAIT FOR ( Cil_Comp_Triplo_A_Rec == FALSE )
            WAIT FOR ( Cil_Comp_Triplo_B_Ava == FALSE )
            WAIT FOR ( Cil_Comp_Triplo_B_Rec == TRUE )
            WAIT FOR ( Cil_Comp_Indiv_Gr_1_Aber == FALSE )
            WAIT FOR ( Cil_Comp_Indiv_Gr_1_Fech == TRUE )
            WAIT FOR ( Cil_Comp_Indiv_Gr_3_Aber == FALSE )
            WAIT FOR ( Cil_Comp_Indiv_Gr_3_Fech == TRUE )
            WAIT FOR ( Cil_Comp_Indiv_Gr_4_Aber == FALSE )
            WAIT FOR ( Cil_Comp_Indiv_Gr_4_Fech == TRUE )
            WAIT FOR ( Cil_Comp_Indiv_Gr_6_Aber == FALSE )
            WAIT FOR ( Cil_Comp_Indiv_Gr_6_Fech == TRUE )
            WAIT FOR ( Cil_1_Gar_1_Ava == TRUE )
            WAIT FOR ( Cil_1_Gar_2_Ava == TRUE )
            WAIT FOR ( Cil_1_Gar_3_Ava == TRUE )
            WAIT FOR ( Cil_1_Gar_4_Ava == TRUE )
            WAIT FOR ( Cil_1_Gar_5_Ava == TRUE )
            WAIT FOR ( Cil_1_Gar_6_Ava == TRUE )
            WAIT FOR ( Cil_2_Gar_1_Ava == TRUE )
            WAIT FOR ( Cil_2_Gar_2_Ava == TRUE )
            WAIT FOR ( Cil_2_Gar_3_Ava == TRUE )
            WAIT FOR ( Cil_2_Gar_4_Ava == TRUE )
            WAIT FOR ( Cil_2_Gar_5_Ava == TRUE )
            WAIT FOR ( Cil_2_Gar_6_Ava == TRUE )

         CASE 161
            Abre_Gar_Triplo_Lado_A = TRUE
            Fecha_Gar_Triplo_Lado_A = FALSE

            Abre_Gar_Triplo_Lado_B = TRUE
            Fecha_Gar_Triplo_Lado_B = FALSE

            Abre_Comp_Indiv_Gar_1 = FALSE
            Fecha_Comp_Indiv_Gar_1 = TRUE

            Abre_Comp_Indiv_Gar_3 = FALSE
            Fecha_Comp_Indiv_Gar_3 = TRUE

            Abre_Comp_Indiv_Gar_4 = FALSE
            Fecha_Comp_Indiv_Gar_4 = TRUE

            Abre_Comp_Indiv_Gar_6 = FALSE
            Fecha_Comp_Indiv_Gar_6 = TRUE

            Ava_Cil_1_Gar_1 = TRUE
            Rec_Cil_1_Gar_1 = FALSE

            Ava_Cil_1_Gar_2 = TRUE
            Rec_Cil_1_Gar_2 = FALSE

            Ava_Cil_1_Gar_3 = TRUE
            Rec_Cil_1_Gar_3 = FALSE

            Ava_Cil_1_Gar_4 = TRUE
            Rec_Cil_1_Gar_4 = FALSE

            Ava_Cil_1_Gar_5 = TRUE
            Rec_Cil_1_Gar_5 = FALSE

            Ava_Cil_1_Gar_6 = TRUE
            Rec_Cil_1_Gar_6 = FALSE

            Ava_Cil_2_Gar_1 = TRUE
            Rec_Cil_2_Gar_1 = FALSE

            Ava_Cil_2_Gar_2 = TRUE
            Rec_Cil_2_Gar_2 = FALSE

            Ava_Cil_2_Gar_3 = TRUE
            Rec_Cil_2_Gar_3 = FALSE

            Ava_Cil_2_Gar_4 = TRUE
            Rec_Cil_2_Gar_4 = FALSE

            Ava_Cil_2_Gar_5 = TRUE
            Rec_Cil_2_Gar_5 = FALSE

            Ava_Cil_2_Gar_6 = TRUE
            Rec_Cil_2_Gar_6 = FALSE

            WAIT FOR ( Cil_Comp_Triplo_A_Ava == TRUE )
            WAIT FOR ( Cil_Comp_Triplo_A_Rec == FALSE )
            WAIT FOR ( Cil_Comp_Triplo_B_Ava == FALSE )
            WAIT FOR ( Cil_Comp_Triplo_B_Rec == TRUE )
            WAIT FOR ( Cil_Comp_Indiv_Gr_1_Aber == FALSE )
            WAIT FOR ( Cil_Comp_Indiv_Gr_1_Fech == TRUE )
            WAIT FOR ( Cil_Comp_Indiv_Gr_3_Aber == FALSE )
            WAIT FOR ( Cil_Comp_Indiv_Gr_3_Fech == TRUE )
            WAIT FOR ( Cil_Comp_Indiv_Gr_4_Aber == FALSE )
            WAIT FOR ( Cil_Comp_Indiv_Gr_4_Fech == TRUE )
            WAIT FOR ( Cil_Comp_Indiv_Gr_6_Aber == FALSE )
            WAIT FOR ( Cil_Comp_Indiv_Gr_6_Fech == TRUE )
            WAIT FOR ( Cil_1_Gar_1_Ava == TRUE )
            WAIT FOR ( Cil_1_Gar_2_Ava == TRUE )
            WAIT FOR ( Cil_1_Gar_3_Ava == TRUE )
            WAIT FOR ( Cil_1_Gar_4_Ava == TRUE )
            WAIT FOR ( Cil_1_Gar_5_Ava == TRUE )
            WAIT FOR ( Cil_1_Gar_6_Ava == TRUE )
            WAIT FOR ( Cil_2_Gar_1_Ava == TRUE )
            WAIT FOR ( Cil_2_Gar_2_Ava == TRUE )
            WAIT FOR ( Cil_2_Gar_3_Ava == TRUE )
            WAIT FOR ( Cil_2_Gar_4_Ava == TRUE )
            WAIT FOR ( Cil_2_Gar_5_Ava == TRUE )
            WAIT FOR ( Cil_2_Gar_6_Ava == TRUE )

         CASE 162
            Abre_Gar_Triplo_Lado_A = TRUE
            Fecha_Gar_Triplo_Lado_A = FALSE

            Abre_Gar_Triplo_Lado_B = TRUE
            Fecha_Gar_Triplo_Lado_B = FALSE

            Abre_Comp_Indiv_Gar_1 = FALSE
            Fecha_Comp_Indiv_Gar_1 = TRUE

            Abre_Comp_Indiv_Gar_3 = FALSE
            Fecha_Comp_Indiv_Gar_3 = TRUE

            Abre_Comp_Indiv_Gar_4 = FALSE
            Fecha_Comp_Indiv_Gar_4 = TRUE

            Abre_Comp_Indiv_Gar_6 = TRUE
            Fecha_Comp_Indiv_Gar_6 = FALSE

            Ava_Cil_1_Gar_1 = TRUE
            Rec_Cil_1_Gar_1 = FALSE

            Ava_Cil_1_Gar_2 = TRUE
            Rec_Cil_1_Gar_2 = FALSE

            Ava_Cil_1_Gar_3 = TRUE
            Rec_Cil_1_Gar_3 = FALSE

            Ava_Cil_1_Gar_4 = TRUE
            Rec_Cil_1_Gar_4 = FALSE

            Ava_Cil_1_Gar_5 = TRUE
            Rec_Cil_1_Gar_5 = FALSE

            Ava_Cil_1_Gar_6 = TRUE
            Rec_Cil_1_Gar_6 = FALSE

            Ava_Cil_2_Gar_1 = TRUE
            Rec_Cil_2_Gar_1 = FALSE

            Ava_Cil_2_Gar_2 = TRUE
            Rec_Cil_2_Gar_2 = FALSE

            Ava_Cil_2_Gar_3 = TRUE
            Rec_Cil_2_Gar_3 = FALSE

            Ava_Cil_2_Gar_4 = TRUE
            Rec_Cil_2_Gar_4 = FALSE

            Ava_Cil_2_Gar_5 = TRUE
            Rec_Cil_2_Gar_5 = FALSE

            Ava_Cil_2_Gar_6 = TRUE
            Rec_Cil_2_Gar_6 = FALSE

            WAIT FOR ( Cil_Comp_Triplo_A_Ava == TRUE )
            WAIT FOR ( Cil_Comp_Triplo_A_Rec == FALSE )
            WAIT FOR ( Cil_Comp_Triplo_B_Ava == TRUE )
            WAIT FOR ( Cil_Comp_Triplo_B_Rec == FALSE )
            WAIT FOR ( Cil_Comp_Indiv_Gr_1_Aber == FALSE )
            WAIT FOR ( Cil_Comp_Indiv_Gr_1_Fech == TRUE )
            WAIT FOR ( Cil_Comp_Indiv_Gr_3_Aber == FALSE )
            WAIT FOR ( Cil_Comp_Indiv_Gr_3_Fech == TRUE )
            WAIT FOR ( Cil_Comp_Indiv_Gr_4_Aber == FALSE )
            WAIT FOR ( Cil_Comp_Indiv_Gr_4_Fech == TRUE )
            WAIT FOR ( Cil_Comp_Indiv_Gr_6_Aber == TRUE )
            WAIT FOR ( Cil_Comp_Indiv_Gr_6_Fech == FALSE )
            WAIT FOR ( Cil_1_Gar_1_Ava == TRUE )
            WAIT FOR ( Cil_1_Gar_2_Ava == TRUE )
            WAIT FOR ( Cil_1_Gar_3_Ava == TRUE )
            WAIT FOR ( Cil_1_Gar_4_Ava == TRUE )
            WAIT FOR ( Cil_1_Gar_5_Ava == TRUE )
            WAIT FOR ( Cil_1_Gar_6_Ava == TRUE )
            WAIT FOR ( Cil_2_Gar_1_Ava == TRUE )
            WAIT FOR ( Cil_2_Gar_2_Ava == TRUE )
            WAIT FOR ( Cil_2_Gar_3_Ava == TRUE )
            WAIT FOR ( Cil_2_Gar_4_Ava == TRUE )
            WAIT FOR ( Cil_2_Gar_5_Ava == TRUE )
            WAIT FOR ( Cil_2_Gar_6_Ava == TRUE )

         CASE 61
            Abre_Gar_Triplo_Lado_A = TRUE
            Fecha_Gar_Triplo_Lado_A = FALSE

            Abre_Gar_Triplo_Lado_B = TRUE
            Fecha_Gar_Triplo_Lado_B = FALSE

            Abre_Comp_Indiv_Gar_1 = TRUE
            Fecha_Comp_Indiv_Gar_1 = FALSE

            Abre_Comp_Indiv_Gar_3 = FALSE
            Fecha_Comp_Indiv_Gar_3 = TRUE

            Abre_Comp_Indiv_Gar_4 = FALSE
            Fecha_Comp_Indiv_Gar_4 = TRUE

            Abre_Comp_Indiv_Gar_6 = TRUE
            Fecha_Comp_Indiv_Gar_6 = FALSE

            Ava_Cil_1_Gar_1 = TRUE
            Rec_Cil_1_Gar_1 = FALSE

            Ava_Cil_1_Gar_2 = TRUE
            Rec_Cil_1_Gar_2 = FALSE

            Ava_Cil_1_Gar_3 = TRUE
            Rec_Cil_1_Gar_3 = FALSE

            Ava_Cil_1_Gar_4 = TRUE
            Rec_Cil_1_Gar_4 = FALSE

            Ava_Cil_1_Gar_5 = TRUE
            Rec_Cil_1_Gar_5 = FALSE

            Ava_Cil_1_Gar_6 = TRUE
            Rec_Cil_1_Gar_6 = FALSE

            Ava_Cil_2_Gar_1 = TRUE
            Rec_Cil_2_Gar_1 = FALSE

            Ava_Cil_2_Gar_2 = TRUE
            Rec_Cil_2_Gar_2 = FALSE

            Ava_Cil_2_Gar_3 = TRUE
            Rec_Cil_2_Gar_3 = FALSE

            Ava_Cil_2_Gar_4 = TRUE
            Rec_Cil_2_Gar_4 = FALSE

            Ava_Cil_2_Gar_5 = TRUE
            Rec_Cil_2_Gar_5 = FALSE

            Ava_Cil_2_Gar_6 = TRUE
            Rec_Cil_2_Gar_6 = FALSE

            WAIT FOR ( Cil_Comp_Triplo_A_Ava == TRUE )
            WAIT FOR ( Cil_Comp_Triplo_A_Rec == FALSE )
            WAIT FOR ( Cil_Comp_Triplo_B_Ava == TRUE )
            WAIT FOR ( Cil_Comp_Triplo_B_Rec == FALSE )
            WAIT FOR ( Cil_Comp_Indiv_Gr_1_Aber == TRUE )
            WAIT FOR ( Cil_Comp_Indiv_Gr_1_Fech == FALSE )
            WAIT FOR ( Cil_Comp_Indiv_Gr_3_Aber == FALSE )
            WAIT FOR ( Cil_Comp_Indiv_Gr_3_Fech == TRUE )
            WAIT FOR ( Cil_Comp_Indiv_Gr_4_Aber == FALSE )
            WAIT FOR ( Cil_Comp_Indiv_Gr_4_Fech == TRUE )
            WAIT FOR ( Cil_Comp_Indiv_Gr_6_Aber == TRUE )
            WAIT FOR ( Cil_Comp_Indiv_Gr_6_Fech == FALSE )
            WAIT FOR ( Cil_1_Gar_1_Ava == TRUE )
            WAIT FOR ( Cil_1_Gar_2_Ava == TRUE )
            WAIT FOR ( Cil_1_Gar_3_Ava == TRUE )
            WAIT FOR ( Cil_1_Gar_4_Ava == TRUE )
            WAIT FOR ( Cil_1_Gar_5_Ava == TRUE )
            WAIT FOR ( Cil_1_Gar_6_Ava == TRUE )
            WAIT FOR ( Cil_2_Gar_1_Ava == TRUE )
            WAIT FOR ( Cil_2_Gar_2_Ava == TRUE )
            WAIT FOR ( Cil_2_Gar_3_Ava == TRUE )
            WAIT FOR ( Cil_2_Gar_4_Ava == TRUE )
            WAIT FOR ( Cil_2_Gar_5_Ava == TRUE )
            WAIT FOR ( Cil_2_Gar_6_Ava == TRUE )

         CASE 62
            Abre_Gar_Triplo_Lado_A = TRUE
            Fecha_Gar_Triplo_Lado_A = FALSE

            Abre_Gar_Triplo_Lado_B = TRUE
            Fecha_Gar_Triplo_Lado_B = FALSE

            Abre_Comp_Indiv_Gar_1 = TRUE
            Fecha_Comp_Indiv_Gar_1 = FALSE

            Abre_Comp_Indiv_Gar_3 = FALSE
            Fecha_Comp_Indiv_Gar_3 = TRUE

            Abre_Comp_Indiv_Gar_4 = FALSE
            Fecha_Comp_Indiv_Gar_4 = TRUE

            Abre_Comp_Indiv_Gar_6 = TRUE
            Fecha_Comp_Indiv_Gar_6 = FALSE

            Ava_Cil_1_Gar_1 = TRUE
            Rec_Cil_1_Gar_1 = FALSE

            Ava_Cil_1_Gar_2 = TRUE
            Rec_Cil_1_Gar_2 = FALSE

            Ava_Cil_1_Gar_3 = TRUE
            Rec_Cil_1_Gar_3 = FALSE

            Ava_Cil_1_Gar_4 = TRUE
            Rec_Cil_1_Gar_4 = FALSE

            Ava_Cil_1_Gar_5 = TRUE
            Rec_Cil_1_Gar_5 = FALSE

            Ava_Cil_1_Gar_6 = TRUE
            Rec_Cil_1_Gar_6 = FALSE

            Ava_Cil_2_Gar_1 = TRUE
            Rec_Cil_2_Gar_1 = FALSE

            Ava_Cil_2_Gar_2 = TRUE
            Rec_Cil_2_Gar_2 = FALSE

            Ava_Cil_2_Gar_3 = TRUE
            Rec_Cil_2_Gar_3 = FALSE

            Ava_Cil_2_Gar_4 = TRUE
            Rec_Cil_2_Gar_4 = FALSE

            Ava_Cil_2_Gar_5 = TRUE
            Rec_Cil_2_Gar_5 = FALSE

            Ava_Cil_2_Gar_6 = TRUE
            Rec_Cil_2_Gar_6 = FALSE

            WAIT FOR ( Cil_Comp_Triplo_A_Ava == TRUE )
            WAIT FOR ( Cil_Comp_Triplo_A_Rec == FALSE )
            WAIT FOR ( Cil_Comp_Triplo_B_Ava == TRUE )
            WAIT FOR ( Cil_Comp_Triplo_B_Rec == FALSE )
            WAIT FOR ( Cil_Comp_Indiv_Gr_1_Aber == TRUE )
            WAIT FOR ( Cil_Comp_Indiv_Gr_1_Fech == FALSE )
            WAIT FOR ( Cil_Comp_Indiv_Gr_3_Aber == FALSE )
            WAIT FOR ( Cil_Comp_Indiv_Gr_3_Fech == TRUE )
            WAIT FOR ( Cil_Comp_Indiv_Gr_4_Aber == FALSE )
            WAIT FOR ( Cil_Comp_Indiv_Gr_4_Fech == TRUE )
            WAIT FOR ( Cil_Comp_Indiv_Gr_6_Aber == TRUE )
            WAIT FOR ( Cil_Comp_Indiv_Gr_6_Fech == FALSE )
            WAIT FOR ( Cil_1_Gar_1_Ava == TRUE )
            WAIT FOR ( Cil_1_Gar_2_Ava == TRUE )
            WAIT FOR ( Cil_1_Gar_3_Ava == TRUE )
            WAIT FOR ( Cil_1_Gar_4_Ava == TRUE )
            WAIT FOR ( Cil_1_Gar_5_Ava == TRUE )
            WAIT FOR ( Cil_1_Gar_6_Ava == TRUE )
            WAIT FOR ( Cil_2_Gar_1_Ava == TRUE )
            WAIT FOR ( Cil_2_Gar_2_Ava == TRUE )
            WAIT FOR ( Cil_2_Gar_3_Ava == TRUE )
            WAIT FOR ( Cil_2_Gar_4_Ava == TRUE )
            WAIT FOR ( Cil_2_Gar_5_Ava == TRUE )
            WAIT FOR ( Cil_2_Gar_6_Ava == TRUE )

         CASE 191
            Abre_Gar_Triplo_Lado_A = TRUE
            Fecha_Gar_Triplo_Lado_A = FALSE

            Abre_Gar_Triplo_Lado_B = TRUE
            Fecha_Gar_Triplo_Lado_B = FALSE

            Abre_Comp_Indiv_Gar_1 = FALSE
            Fecha_Comp_Indiv_Gar_1 = TRUE

            Abre_Comp_Indiv_Gar_3 = FALSE
            Fecha_Comp_Indiv_Gar_3 = TRUE

            Abre_Comp_Indiv_Gar_4 = FALSE
            Fecha_Comp_Indiv_Gar_4 = TRUE

            Abre_Comp_Indiv_Gar_6 = FALSE
            Fecha_Comp_Indiv_Gar_6 = TRUE

            Ava_Cil_1_Gar_1 = TRUE
            Rec_Cil_1_Gar_1 = FALSE

            Ava_Cil_1_Gar_2 = TRUE
            Rec_Cil_1_Gar_2 = FALSE

            Ava_Cil_1_Gar_3 = TRUE
            Rec_Cil_1_Gar_3 = FALSE

            Ava_Cil_1_Gar_4 = TRUE
            Rec_Cil_1_Gar_4 = FALSE

            Ava_Cil_1_Gar_5 = TRUE
            Rec_Cil_1_Gar_5 = FALSE

            Ava_Cil_1_Gar_6 = TRUE
            Rec_Cil_1_Gar_6 = FALSE

            Ava_Cil_2_Gar_1 = TRUE
            Rec_Cil_2_Gar_1 = FALSE

            Ava_Cil_2_Gar_2 = TRUE
            Rec_Cil_2_Gar_2 = FALSE

            Ava_Cil_2_Gar_3 = TRUE
            Rec_Cil_2_Gar_3 = FALSE

            Ava_Cil_2_Gar_4 = TRUE
            Rec_Cil_2_Gar_4 = FALSE

            Ava_Cil_2_Gar_5 = TRUE
            Rec_Cil_2_Gar_5 = FALSE

            Ava_Cil_2_Gar_6 = TRUE
            Rec_Cil_2_Gar_6 = FALSE

            WAIT FOR ( Cil_Comp_Triplo_A_Ava == TRUE )
            WAIT FOR ( Cil_Comp_Triplo_A_Rec == FALSE )
            WAIT FOR ( Cil_Comp_Triplo_B_Ava == TRUE )
            WAIT FOR ( Cil_Comp_Triplo_B_Rec == FALSE )
            WAIT FOR ( Cil_Comp_Indiv_Gr_1_Aber == FALSE )
            WAIT FOR ( Cil_Comp_Indiv_Gr_1_Fech == TRUE )
            WAIT FOR ( Cil_Comp_Indiv_Gr_3_Aber == FALSE )
            WAIT FOR ( Cil_Comp_Indiv_Gr_3_Fech == TRUE )
            WAIT FOR ( Cil_Comp_Indiv_Gr_4_Aber == FALSE )
            WAIT FOR ( Cil_Comp_Indiv_Gr_4_Fech == TRUE )
            WAIT FOR ( Cil_Comp_Indiv_Gr_6_Aber == FALSE )
            WAIT FOR ( Cil_Comp_Indiv_Gr_6_Fech == TRUE )
            WAIT FOR ( Cil_1_Gar_1_Ava == TRUE )
            WAIT FOR ( Cil_1_Gar_2_Ava == TRUE )
            WAIT FOR ( Cil_1_Gar_3_Ava == TRUE )
            WAIT FOR ( Cil_1_Gar_4_Ava == TRUE )
            WAIT FOR ( Cil_1_Gar_5_Ava == TRUE )
            WAIT FOR ( Cil_1_Gar_6_Ava == TRUE )
            WAIT FOR ( Cil_2_Gar_1_Ava == TRUE )
            WAIT FOR ( Cil_2_Gar_2_Ava == TRUE )
            WAIT FOR ( Cil_2_Gar_3_Ava == TRUE )
            WAIT FOR ( Cil_2_Gar_4_Ava == TRUE )
            WAIT FOR ( Cil_2_Gar_5_Ava == TRUE )
            WAIT FOR ( Cil_2_Gar_6_Ava == TRUE )

         CASE 192
            Abre_Gar_Triplo_Lado_A = TRUE
            Fecha_Gar_Triplo_Lado_A = FALSE

            Abre_Gar_Triplo_Lado_B = TRUE
            Fecha_Gar_Triplo_Lado_B = FALSE

            Abre_Comp_Indiv_Gar_1 = FALSE
            Fecha_Comp_Indiv_Gar_1 = TRUE

            Abre_Comp_Indiv_Gar_3 = FALSE
            Fecha_Comp_Indiv_Gar_3 = TRUE

            Abre_Comp_Indiv_Gar_4 = FALSE
            Fecha_Comp_Indiv_Gar_4 = TRUE

            Abre_Comp_Indiv_Gar_6 = FALSE
            Fecha_Comp_Indiv_Gar_6 = TRUE

            Ava_Cil_1_Gar_1 = TRUE
            Rec_Cil_1_Gar_1 = FALSE

            Ava_Cil_1_Gar_2 = TRUE
            Rec_Cil_1_Gar_2 = FALSE

            Ava_Cil_1_Gar_3 = TRUE
            Rec_Cil_1_Gar_3 = FALSE

            Ava_Cil_1_Gar_4 = TRUE
            Rec_Cil_1_Gar_4 = FALSE

            Ava_Cil_1_Gar_5 = TRUE
            Rec_Cil_1_Gar_5 = FALSE

            Ava_Cil_1_Gar_6 = TRUE
            Rec_Cil_1_Gar_6 = FALSE

            Ava_Cil_2_Gar_1 = TRUE
            Rec_Cil_2_Gar_1 = FALSE

            Ava_Cil_2_Gar_2 = TRUE
            Rec_Cil_2_Gar_2 = FALSE

            Ava_Cil_2_Gar_3 = TRUE
            Rec_Cil_2_Gar_3 = FALSE

            Ava_Cil_2_Gar_4 = TRUE
            Rec_Cil_2_Gar_4 = FALSE

            Ava_Cil_2_Gar_5 = TRUE
            Rec_Cil_2_Gar_5 = FALSE

            Ava_Cil_2_Gar_6 = TRUE
            Rec_Cil_2_Gar_6 = FALSE

            WAIT FOR ( Cil_Comp_Triplo_A_Ava == TRUE )
            WAIT FOR ( Cil_Comp_Triplo_A_Rec == FALSE )
            WAIT FOR ( Cil_Comp_Triplo_B_Ava == TRUE )
            WAIT FOR ( Cil_Comp_Triplo_B_Rec == FALSE )
            WAIT FOR ( Cil_Comp_Indiv_Gr_1_Aber == FALSE )
            WAIT FOR ( Cil_Comp_Indiv_Gr_1_Fech == TRUE )
            WAIT FOR ( Cil_Comp_Indiv_Gr_3_Aber == FALSE )
            WAIT FOR ( Cil_Comp_Indiv_Gr_3_Fech == TRUE )
            WAIT FOR ( Cil_Comp_Indiv_Gr_4_Aber == FALSE )
            WAIT FOR ( Cil_Comp_Indiv_Gr_4_Fech == TRUE )
            WAIT FOR ( Cil_Comp_Indiv_Gr_6_Aber == FALSE )
            WAIT FOR ( Cil_Comp_Indiv_Gr_6_Fech == TRUE )
            WAIT FOR ( Cil_1_Gar_1_Ava == TRUE )
            WAIT FOR ( Cil_1_Gar_2_Ava == TRUE )
            WAIT FOR ( Cil_1_Gar_3_Ava == TRUE )
            WAIT FOR ( Cil_1_Gar_4_Ava == TRUE )
            WAIT FOR ( Cil_1_Gar_5_Ava == TRUE )
            WAIT FOR ( Cil_1_Gar_6_Ava == TRUE )
            WAIT FOR ( Cil_2_Gar_1_Ava == TRUE )
            WAIT FOR ( Cil_2_Gar_2_Ava == TRUE )
            WAIT FOR ( Cil_2_Gar_3_Ava == TRUE )
            WAIT FOR ( Cil_2_Gar_4_Ava == TRUE )
            WAIT FOR ( Cil_2_Gar_5_Ava == TRUE )
            WAIT FOR ( Cil_2_Gar_6_Ava == TRUE )

         CASE 81
            Abre_Gar_Triplo_Lado_A = TRUE
            Fecha_Gar_Triplo_Lado_A = FALSE

            Abre_Gar_Triplo_Lado_B = TRUE
            Fecha_Gar_Triplo_Lado_B = FALSE

            Abre_Comp_Indiv_Gar_1 = FALSE
            Fecha_Comp_Indiv_Gar_1 = TRUE

            Abre_Comp_Indiv_Gar_3 = FALSE
            Fecha_Comp_Indiv_Gar_3 = TRUE

            Abre_Comp_Indiv_Gar_4 = FALSE
            Fecha_Comp_Indiv_Gar_4 = TRUE

            Abre_Comp_Indiv_Gar_6 = TRUE
            Fecha_Comp_Indiv_Gar_6 = FALSE

            Ava_Cil_1_Gar_1 = TRUE
            Rec_Cil_1_Gar_1 = FALSE

            Ava_Cil_1_Gar_2 = TRUE
            Rec_Cil_1_Gar_2 = FALSE

            Ava_Cil_1_Gar_3 = TRUE
            Rec_Cil_1_Gar_3 = FALSE

            Ava_Cil_1_Gar_4 = TRUE
            Rec_Cil_1_Gar_4 = FALSE

            Ava_Cil_1_Gar_5 = TRUE
            Rec_Cil_1_Gar_5 = FALSE

            Ava_Cil_1_Gar_6 = TRUE
            Rec_Cil_1_Gar_6 = FALSE

            Ava_Cil_2_Gar_1 = TRUE
            Rec_Cil_2_Gar_1 = FALSE

            Ava_Cil_2_Gar_2 = TRUE
            Rec_Cil_2_Gar_2 = FALSE

            Ava_Cil_2_Gar_3 = TRUE
            Rec_Cil_2_Gar_3 = FALSE

            Ava_Cil_2_Gar_4 = TRUE
            Rec_Cil_2_Gar_4 = FALSE

            Ava_Cil_2_Gar_5 = TRUE
            Rec_Cil_2_Gar_5 = FALSE

            Ava_Cil_2_Gar_6 = TRUE
            Rec_Cil_2_Gar_6 = FALSE

            WAIT FOR ( Cil_Comp_Triplo_A_Ava == TRUE )
            WAIT FOR ( Cil_Comp_Triplo_A_Rec == FALSE )
            WAIT FOR ( Cil_Comp_Triplo_B_Ava == TRUE )
            WAIT FOR ( Cil_Comp_Triplo_B_Rec == FALSE )
            WAIT FOR ( Cil_Comp_Indiv_Gr_1_Aber == FALSE )
            WAIT FOR ( Cil_Comp_Indiv_Gr_1_Fech == TRUE )
            WAIT FOR ( Cil_Comp_Indiv_Gr_3_Aber == FALSE )
            WAIT FOR ( Cil_Comp_Indiv_Gr_3_Fech == TRUE )
            WAIT FOR ( Cil_Comp_Indiv_Gr_4_Aber == FALSE )
            WAIT FOR ( Cil_Comp_Indiv_Gr_4_Fech == TRUE )
            WAIT FOR ( Cil_Comp_Indiv_Gr_6_Aber == TRUE )
            WAIT FOR ( Cil_Comp_Indiv_Gr_6_Fech == FALSE )
            WAIT FOR ( Cil_1_Gar_1_Ava == TRUE )
            WAIT FOR ( Cil_1_Gar_2_Ava == TRUE )
            WAIT FOR ( Cil_1_Gar_3_Ava == TRUE )
            WAIT FOR ( Cil_1_Gar_4_Ava == TRUE )
            WAIT FOR ( Cil_1_Gar_5_Ava == TRUE )
            WAIT FOR ( Cil_1_Gar_6_Ava == TRUE )
            WAIT FOR ( Cil_2_Gar_1_Ava == TRUE )
            WAIT FOR ( Cil_2_Gar_2_Ava == TRUE )
            WAIT FOR ( Cil_2_Gar_3_Ava == TRUE )
            WAIT FOR ( Cil_2_Gar_4_Ava == TRUE )
            WAIT FOR ( Cil_2_Gar_5_Ava == TRUE )
            WAIT FOR ( Cil_2_Gar_6_Ava == TRUE )

         CASE 82
            Abre_Gar_Triplo_Lado_A = TRUE
            Fecha_Gar_Triplo_Lado_A = FALSE

            Abre_Gar_Triplo_Lado_B = TRUE
            Fecha_Gar_Triplo_Lado_B = FALSE

            Abre_Comp_Indiv_Gar_1 = FALSE
            Fecha_Comp_Indiv_Gar_1 = TRUE

            Abre_Comp_Indiv_Gar_3 = TRUE
            Fecha_Comp_Indiv_Gar_3 = FALSE

            Abre_Comp_Indiv_Gar_4 = TRUE
            Fecha_Comp_Indiv_Gar_4 = FALSE

            Abre_Comp_Indiv_Gar_6 = FALSE
            Fecha_Comp_Indiv_Gar_6 = TRUE

            Ava_Cil_1_Gar_1 = TRUE
            Rec_Cil_1_Gar_1 = FALSE

            Ava_Cil_1_Gar_2 = TRUE
            Rec_Cil_1_Gar_2 = FALSE

            Ava_Cil_1_Gar_3 = TRUE
            Rec_Cil_1_Gar_3 = FALSE

            Ava_Cil_1_Gar_4 = TRUE
            Rec_Cil_1_Gar_4 = FALSE

            Ava_Cil_1_Gar_5 = TRUE
            Rec_Cil_1_Gar_5 = FALSE

            Ava_Cil_1_Gar_6 = TRUE
            Rec_Cil_1_Gar_6 = FALSE

            Ava_Cil_2_Gar_1 = TRUE
            Rec_Cil_2_Gar_1 = FALSE

            Ava_Cil_2_Gar_2 = TRUE
            Rec_Cil_2_Gar_2 = FALSE

            Ava_Cil_2_Gar_3 = TRUE
            Rec_Cil_2_Gar_3 = FALSE

            Ava_Cil_2_Gar_4 = TRUE
            Rec_Cil_2_Gar_4 = FALSE

            Ava_Cil_2_Gar_5 = TRUE
            Rec_Cil_2_Gar_5 = FALSE

            Ava_Cil_2_Gar_6 = TRUE
            Rec_Cil_2_Gar_6 = FALSE

            WAIT FOR ( Cil_Comp_Triplo_A_Ava == FALSE )
            WAIT FOR ( Cil_Comp_Triplo_A_Rec == TRUE )
            WAIT FOR ( Cil_Comp_Triplo_B_Ava == FALSE )
            WAIT FOR ( Cil_Comp_Triplo_B_Rec == TRUE )
            WAIT FOR ( Cil_Comp_Indiv_Gr_1_Aber == FALSE )
            WAIT FOR ( Cil_Comp_Indiv_Gr_1_Fech == TRUE )
            WAIT FOR ( Cil_Comp_Indiv_Gr_3_Aber == TRUE )
            WAIT FOR ( Cil_Comp_Indiv_Gr_3_Fech == FALSE )
            WAIT FOR ( Cil_Comp_Indiv_Gr_4_Aber == TRUE )
            WAIT FOR ( Cil_Comp_Indiv_Gr_4_Fech == FALSE )
            WAIT FOR ( Cil_Comp_Indiv_Gr_6_Aber == FALSE )
            WAIT FOR ( Cil_Comp_Indiv_Gr_6_Fech == TRUE )
            WAIT FOR ( Cil_1_Gar_1_Ava == TRUE )
            WAIT FOR ( Cil_1_Gar_2_Ava == TRUE )
            WAIT FOR ( Cil_1_Gar_3_Ava == TRUE )
            WAIT FOR ( Cil_1_Gar_4_Ava == TRUE )
            WAIT FOR ( Cil_1_Gar_5_Ava == TRUE )
            WAIT FOR ( Cil_1_Gar_6_Ava == TRUE )
            WAIT FOR ( Cil_2_Gar_1_Ava == TRUE )
            WAIT FOR ( Cil_2_Gar_2_Ava == TRUE )
            WAIT FOR ( Cil_2_Gar_3_Ava == TRUE )
            WAIT FOR ( Cil_2_Gar_4_Ava == TRUE )
            WAIT FOR ( Cil_2_Gar_5_Ava == TRUE )
            WAIT FOR ( Cil_2_Gar_6_Ava == TRUE )

         CASE 91
            Abre_Gar_Triplo_Lado_A = TRUE
            Fecha_Gar_Triplo_Lado_A = FALSE

            Abre_Gar_Triplo_Lado_B = TRUE
            Fecha_Gar_Triplo_Lado_B = FALSE

            Abre_Comp_Indiv_Gar_1 = FALSE
            Fecha_Comp_Indiv_Gar_1 = TRUE

            Abre_Comp_Indiv_Gar_3 = TRUE
            Fecha_Comp_Indiv_Gar_3 = FALSE

            Abre_Comp_Indiv_Gar_4 = TRUE
            Fecha_Comp_Indiv_Gar_4 = FALSE

            Abre_Comp_Indiv_Gar_6 = FALSE
            Fecha_Comp_Indiv_Gar_6 = TRUE

            Ava_Cil_1_Gar_1 = TRUE
            Rec_Cil_1_Gar_1 = FALSE

            Ava_Cil_1_Gar_2 = TRUE
            Rec_Cil_1_Gar_2 = FALSE

            Ava_Cil_1_Gar_3 = TRUE
            Rec_Cil_1_Gar_3 = FALSE

            Ava_Cil_1_Gar_4 = TRUE
            Rec_Cil_1_Gar_4 = FALSE

            Ava_Cil_1_Gar_5 = TRUE
            Rec_Cil_1_Gar_5 = FALSE

            Ava_Cil_1_Gar_6 = TRUE
            Rec_Cil_1_Gar_6 = FALSE

            Ava_Cil_2_Gar_1 = TRUE
            Rec_Cil_2_Gar_1 = FALSE

            Ava_Cil_2_Gar_2 = TRUE
            Rec_Cil_2_Gar_2 = FALSE

            Ava_Cil_2_Gar_3 = TRUE
            Rec_Cil_2_Gar_3 = FALSE

            Ava_Cil_2_Gar_4 = TRUE
            Rec_Cil_2_Gar_4 = FALSE

            Ava_Cil_2_Gar_5 = TRUE
            Rec_Cil_2_Gar_5 = FALSE

            Ava_Cil_2_Gar_6 = TRUE
            Rec_Cil_2_Gar_6 = FALSE

            WAIT FOR ( Cil_Comp_Triplo_A_Ava == FALSE )
            WAIT FOR ( Cil_Comp_Triplo_A_Rec == TRUE )
            WAIT FOR ( Cil_Comp_Triplo_B_Ava == FALSE )
            WAIT FOR ( Cil_Comp_Triplo_B_Rec == TRUE )
            WAIT FOR ( Cil_Comp_Indiv_Gr_1_Aber == FALSE )
            WAIT FOR ( Cil_Comp_Indiv_Gr_1_Fech == TRUE )
            WAIT FOR ( Cil_Comp_Indiv_Gr_3_Aber == TRUE )
            WAIT FOR ( Cil_Comp_Indiv_Gr_3_Fech == FALSE )
            WAIT FOR ( Cil_Comp_Indiv_Gr_4_Aber == TRUE )
            WAIT FOR ( Cil_Comp_Indiv_Gr_4_Fech == FALSE )
            WAIT FOR ( Cil_Comp_Indiv_Gr_6_Aber == FALSE )
            WAIT FOR ( Cil_Comp_Indiv_Gr_6_Fech == TRUE )
            WAIT FOR ( Cil_1_Gar_1_Ava == TRUE )
            WAIT FOR ( Cil_1_Gar_2_Ava == TRUE )
            WAIT FOR ( Cil_1_Gar_3_Ava == TRUE )
            WAIT FOR ( Cil_1_Gar_4_Ava == TRUE )
            WAIT FOR ( Cil_1_Gar_5_Ava == TRUE )
            WAIT FOR ( Cil_1_Gar_6_Ava == TRUE )
            WAIT FOR ( Cil_2_Gar_1_Ava == TRUE )
            WAIT FOR ( Cil_2_Gar_2_Ava == TRUE )
            WAIT FOR ( Cil_2_Gar_3_Ava == TRUE )
            WAIT FOR ( Cil_2_Gar_4_Ava == TRUE )
            WAIT FOR ( Cil_2_Gar_5_Ava == TRUE )
            WAIT FOR ( Cil_2_Gar_6_Ava == TRUE )

         CASE 92
            Abre_Gar_Triplo_Lado_A = TRUE
            Fecha_Gar_Triplo_Lado_A = FALSE

            Abre_Gar_Triplo_Lado_B = TRUE
            Fecha_Gar_Triplo_Lado_B = FALSE

            Abre_Comp_Indiv_Gar_1 = FALSE
            Fecha_Comp_Indiv_Gar_1 = TRUE

            Abre_Comp_Indiv_Gar_3 = FALSE
            Fecha_Comp_Indiv_Gar_3 = TRUE

            Abre_Comp_Indiv_Gar_4 = FALSE
            Fecha_Comp_Indiv_Gar_4 = TRUE

            Abre_Comp_Indiv_Gar_6 = TRUE
            Fecha_Comp_Indiv_Gar_6 = FALSE

            Ava_Cil_1_Gar_1 = TRUE
            Rec_Cil_1_Gar_1 = FALSE

            Ava_Cil_1_Gar_2 = TRUE
            Rec_Cil_1_Gar_2 = FALSE

            Ava_Cil_1_Gar_3 = TRUE
            Rec_Cil_1_Gar_3 = FALSE

            Ava_Cil_1_Gar_4 = TRUE
            Rec_Cil_1_Gar_4 = FALSE

            Ava_Cil_1_Gar_5 = TRUE
            Rec_Cil_1_Gar_5 = FALSE

            Ava_Cil_1_Gar_6 = TRUE
            Rec_Cil_1_Gar_6 = FALSE

            Ava_Cil_2_Gar_1 = TRUE
            Rec_Cil_2_Gar_1 = FALSE

            Ava_Cil_2_Gar_2 = TRUE
            Rec_Cil_2_Gar_2 = FALSE

            Ava_Cil_2_Gar_3 = TRUE
            Rec_Cil_2_Gar_3 = FALSE

            Ava_Cil_2_Gar_4 = TRUE
            Rec_Cil_2_Gar_4 = FALSE

            Ava_Cil_2_Gar_5 = TRUE
            Rec_Cil_2_Gar_5 = FALSE

            Ava_Cil_2_Gar_6 = TRUE
            Rec_Cil_2_Gar_6 = FALSE

            WAIT FOR ( Cil_Comp_Triplo_A_Ava == TRUE )
            WAIT FOR ( Cil_Comp_Triplo_A_Rec == FALSE )
            WAIT FOR ( Cil_Comp_Triplo_B_Ava == TRUE )
            WAIT FOR ( Cil_Comp_Triplo_B_Rec == FALSE )
            WAIT FOR ( Cil_Comp_Indiv_Gr_1_Aber == FALSE )
            WAIT FOR ( Cil_Comp_Indiv_Gr_1_Fech == TRUE )
            WAIT FOR ( Cil_Comp_Indiv_Gr_3_Aber == FALSE )
            WAIT FOR ( Cil_Comp_Indiv_Gr_3_Fech == TRUE )
            WAIT FOR ( Cil_Comp_Indiv_Gr_4_Aber == FALSE )
            WAIT FOR ( Cil_Comp_Indiv_Gr_4_Fech == TRUE )
            WAIT FOR ( Cil_Comp_Indiv_Gr_6_Aber == TRUE )
            WAIT FOR ( Cil_Comp_Indiv_Gr_6_Fech == FALSE )
            WAIT FOR ( Cil_1_Gar_1_Ava == TRUE )
            WAIT FOR ( Cil_1_Gar_2_Ava == TRUE )
            WAIT FOR ( Cil_1_Gar_3_Ava == TRUE )
            WAIT FOR ( Cil_1_Gar_4_Ava == TRUE )
            WAIT FOR ( Cil_1_Gar_5_Ava == TRUE )
            WAIT FOR ( Cil_1_Gar_6_Ava == TRUE )
            WAIT FOR ( Cil_2_Gar_1_Ava == TRUE )
            WAIT FOR ( Cil_2_Gar_2_Ava == TRUE )
            WAIT FOR ( Cil_2_Gar_3_Ava == TRUE )
            WAIT FOR ( Cil_2_Gar_4_Ava == TRUE )
            WAIT FOR ( Cil_2_Gar_5_Ava == TRUE )
            WAIT FOR ( Cil_2_Gar_6_Ava == TRUE )

         CASE 151
            Abre_Gar_Triplo_Lado_A = TRUE
            Fecha_Gar_Triplo_Lado_A = FALSE

            Abre_Gar_Triplo_Lado_B = TRUE
            Fecha_Gar_Triplo_Lado_B = FALSE

            Abre_Comp_Indiv_Gar_1 = TRUE
            Fecha_Comp_Indiv_Gar_1 = FALSE

            Abre_Comp_Indiv_Gar_3 = FALSE
            Fecha_Comp_Indiv_Gar_3 = TRUE

            Abre_Comp_Indiv_Gar_4 = FALSE
            Fecha_Comp_Indiv_Gar_4 = TRUE

            Abre_Comp_Indiv_Gar_6 = TRUE
            Fecha_Comp_Indiv_Gar_6 = FALSE

            Ava_Cil_1_Gar_1 = TRUE
            Rec_Cil_1_Gar_1 = FALSE

            Ava_Cil_1_Gar_2 = TRUE
            Rec_Cil_1_Gar_2 = FALSE

            Ava_Cil_1_Gar_3 = TRUE
            Rec_Cil_1_Gar_3 = FALSE

            Ava_Cil_1_Gar_4 = TRUE
            Rec_Cil_1_Gar_4 = FALSE

            Ava_Cil_1_Gar_5 = TRUE
            Rec_Cil_1_Gar_5 = FALSE

            Ava_Cil_1_Gar_6 = TRUE
            Rec_Cil_1_Gar_6 = FALSE

            Ava_Cil_2_Gar_1 = TRUE
            Rec_Cil_2_Gar_1 = FALSE

            Ava_Cil_2_Gar_2 = TRUE
            Rec_Cil_2_Gar_2 = FALSE

            Ava_Cil_2_Gar_3 = TRUE
            Rec_Cil_2_Gar_3 = FALSE

            Ava_Cil_2_Gar_4 = TRUE
            Rec_Cil_2_Gar_4 = FALSE

            Ava_Cil_2_Gar_5 = TRUE
            Rec_Cil_2_Gar_5 = FALSE

            Ava_Cil_2_Gar_6 = TRUE
            Rec_Cil_2_Gar_6 = FALSE

            WAIT FOR ( Cil_Comp_Triplo_A_Ava == TRUE )
            WAIT FOR ( Cil_Comp_Triplo_A_Rec == FALSE )
            WAIT FOR ( Cil_Comp_Triplo_B_Ava == TRUE )
            WAIT FOR ( Cil_Comp_Triplo_B_Rec == FALSE )
            WAIT FOR ( Cil_Comp_Indiv_Gr_1_Aber == TRUE )
            WAIT FOR ( Cil_Comp_Indiv_Gr_1_Fech == FALSE )
            WAIT FOR ( Cil_Comp_Indiv_Gr_3_Aber == FALSE )
            WAIT FOR ( Cil_Comp_Indiv_Gr_3_Fech == TRUE )
            WAIT FOR ( Cil_Comp_Indiv_Gr_4_Aber == FALSE )
            WAIT FOR ( Cil_Comp_Indiv_Gr_4_Fech == TRUE )
            WAIT FOR ( Cil_Comp_Indiv_Gr_6_Aber == TRUE )
            WAIT FOR ( Cil_Comp_Indiv_Gr_6_Fech == FALSE )
            WAIT FOR ( Cil_1_Gar_1_Ava == TRUE )
            WAIT FOR ( Cil_1_Gar_2_Ava == TRUE )
            WAIT FOR ( Cil_1_Gar_3_Ava == TRUE )
            WAIT FOR ( Cil_1_Gar_4_Ava == TRUE )
            WAIT FOR ( Cil_1_Gar_5_Ava == TRUE )
            WAIT FOR ( Cil_1_Gar_6_Ava == TRUE )
            WAIT FOR ( Cil_2_Gar_1_Ava == TRUE )
            WAIT FOR ( Cil_2_Gar_2_Ava == TRUE )
            WAIT FOR ( Cil_2_Gar_3_Ava == TRUE )
            WAIT FOR ( Cil_2_Gar_4_Ava == TRUE )
            WAIT FOR ( Cil_2_Gar_5_Ava == TRUE )
            WAIT FOR ( Cil_2_Gar_6_Ava == TRUE )

         CASE 141
            Abre_Gar_Triplo_Lado_A = TRUE
            Fecha_Gar_Triplo_Lado_A = FALSE

            Abre_Gar_Triplo_Lado_B = TRUE
            Fecha_Gar_Triplo_Lado_B = FALSE

            Abre_Comp_Indiv_Gar_1 = FALSE
            Fecha_Comp_Indiv_Gar_1 = TRUE

            Abre_Comp_Indiv_Gar_3 = FALSE
            Fecha_Comp_Indiv_Gar_3 = TRUE

            Abre_Comp_Indiv_Gar_4 = FALSE
            Fecha_Comp_Indiv_Gar_4 = TRUE

            Abre_Comp_Indiv_Gar_6 = FALSE
            Fecha_Comp_Indiv_Gar_6 = TRUE

            Ava_Cil_1_Gar_1 = TRUE
            Rec_Cil_1_Gar_1 = FALSE

            Ava_Cil_1_Gar_2 = TRUE
            Rec_Cil_1_Gar_2 = FALSE

            Ava_Cil_1_Gar_3 = TRUE
            Rec_Cil_1_Gar_3 = FALSE

            Ava_Cil_1_Gar_4 = TRUE
            Rec_Cil_1_Gar_4 = FALSE

            Ava_Cil_1_Gar_5 = TRUE
            Rec_Cil_1_Gar_5 = FALSE

            Ava_Cil_1_Gar_6 = TRUE
            Rec_Cil_1_Gar_6 = FALSE

            Ava_Cil_2_Gar_1 = TRUE
            Rec_Cil_2_Gar_1 = FALSE

            Ava_Cil_2_Gar_2 = TRUE
            Rec_Cil_2_Gar_2 = FALSE

            Ava_Cil_2_Gar_3 = TRUE
            Rec_Cil_2_Gar_3 = FALSE

            Ava_Cil_2_Gar_4 = TRUE
            Rec_Cil_2_Gar_4 = FALSE

            Ava_Cil_2_Gar_5 = TRUE
            Rec_Cil_2_Gar_5 = FALSE

            Ava_Cil_2_Gar_6 = TRUE
            Rec_Cil_2_Gar_6 = FALSE

            WAIT FOR ( Cil_Comp_Triplo_A_Ava == FALSE )
            WAIT FOR ( Cil_Comp_Triplo_A_Rec == TRUE )
            WAIT FOR ( Cil_Comp_Triplo_B_Ava == FALSE )
            WAIT FOR ( Cil_Comp_Triplo_B_Rec == TRUE )
            WAIT FOR ( Cil_Comp_Indiv_Gr_1_Aber == FALSE )
            WAIT FOR ( Cil_Comp_Indiv_Gr_1_Fech == TRUE )
            WAIT FOR ( Cil_Comp_Indiv_Gr_3_Aber == FALSE )
            WAIT FOR ( Cil_Comp_Indiv_Gr_3_Fech == TRUE )
            WAIT FOR ( Cil_Comp_Indiv_Gr_4_Aber == FALSE )
            WAIT FOR ( Cil_Comp_Indiv_Gr_4_Fech == TRUE )
            WAIT FOR ( Cil_Comp_Indiv_Gr_6_Aber == FALSE )
            WAIT FOR ( Cil_Comp_Indiv_Gr_6_Fech == TRUE )
            WAIT FOR ( Cil_1_Gar_1_Ava == TRUE )
            WAIT FOR ( Cil_1_Gar_2_Ava == TRUE )
            WAIT FOR ( Cil_1_Gar_3_Ava == TRUE )
            WAIT FOR ( Cil_1_Gar_4_Ava == TRUE )
            WAIT FOR ( Cil_1_Gar_5_Ava == TRUE )
            WAIT FOR ( Cil_1_Gar_6_Ava == TRUE )
            WAIT FOR ( Cil_2_Gar_1_Ava == TRUE )
            WAIT FOR ( Cil_2_Gar_2_Ava == TRUE )
            WAIT FOR ( Cil_2_Gar_3_Ava == TRUE )
            WAIT FOR ( Cil_2_Gar_4_Ava == TRUE )
            WAIT FOR ( Cil_2_Gar_5_Ava == TRUE )
            WAIT FOR ( Cil_2_Gar_6_Ava == TRUE )

         CASE 142
            Abre_Gar_Triplo_Lado_A = TRUE
            Fecha_Gar_Triplo_Lado_A = FALSE

            Abre_Gar_Triplo_Lado_B = TRUE
            Fecha_Gar_Triplo_Lado_B = FALSE

            Abre_Comp_Indiv_Gar_1 = FALSE
            Fecha_Comp_Indiv_Gar_1 = TRUE

            Abre_Comp_Indiv_Gar_3 = FALSE
            Fecha_Comp_Indiv_Gar_3 = TRUE

            Abre_Comp_Indiv_Gar_4 = FALSE
            Fecha_Comp_Indiv_Gar_4 = TRUE

            Abre_Comp_Indiv_Gar_6 = FALSE
            Fecha_Comp_Indiv_Gar_6 = TRUE

            Ava_Cil_1_Gar_1 = TRUE
            Rec_Cil_1_Gar_1 = FALSE

            Ava_Cil_1_Gar_2 = TRUE
            Rec_Cil_1_Gar_2 = FALSE

            Ava_Cil_1_Gar_3 = TRUE
            Rec_Cil_1_Gar_3 = FALSE

            Ava_Cil_1_Gar_4 = TRUE
            Rec_Cil_1_Gar_4 = FALSE

            Ava_Cil_1_Gar_5 = TRUE
            Rec_Cil_1_Gar_5 = FALSE

            Ava_Cil_1_Gar_6 = TRUE
            Rec_Cil_1_Gar_6 = FALSE

            Ava_Cil_2_Gar_1 = TRUE
            Rec_Cil_2_Gar_1 = FALSE

            Ava_Cil_2_Gar_2 = TRUE
            Rec_Cil_2_Gar_2 = FALSE

            Ava_Cil_2_Gar_3 = TRUE
            Rec_Cil_2_Gar_3 = FALSE

            Ava_Cil_2_Gar_4 = TRUE
            Rec_Cil_2_Gar_4 = FALSE

            Ava_Cil_2_Gar_5 = TRUE
            Rec_Cil_2_Gar_5 = FALSE

            Ava_Cil_2_Gar_6 = TRUE
            Rec_Cil_2_Gar_6 = FALSE

            WAIT FOR ( Cil_Comp_Triplo_A_Ava == FALSE )
            WAIT FOR ( Cil_Comp_Triplo_A_Rec == TRUE )
            WAIT FOR ( Cil_Comp_Triplo_B_Ava == FALSE )
            WAIT FOR ( Cil_Comp_Triplo_B_Rec == TRUE )
            WAIT FOR ( Cil_Comp_Indiv_Gr_1_Aber == FALSE )
            WAIT FOR ( Cil_Comp_Indiv_Gr_1_Fech == TRUE )
            WAIT FOR ( Cil_Comp_Indiv_Gr_3_Aber == FALSE )
            WAIT FOR ( Cil_Comp_Indiv_Gr_3_Fech == TRUE )
            WAIT FOR ( Cil_Comp_Indiv_Gr_4_Aber == FALSE )
            WAIT FOR ( Cil_Comp_Indiv_Gr_4_Fech == TRUE )
            WAIT FOR ( Cil_Comp_Indiv_Gr_6_Aber == FALSE )
            WAIT FOR ( Cil_Comp_Indiv_Gr_6_Fech == TRUE )
            WAIT FOR ( Cil_1_Gar_1_Ava == TRUE )
            WAIT FOR ( Cil_1_Gar_2_Ava == TRUE )
            WAIT FOR ( Cil_1_Gar_3_Ava == TRUE )
            WAIT FOR ( Cil_1_Gar_4_Ava == TRUE )
            WAIT FOR ( Cil_1_Gar_5_Ava == TRUE )
            WAIT FOR ( Cil_1_Gar_6_Ava == TRUE )
            WAIT FOR ( Cil_2_Gar_1_Ava == TRUE )
            WAIT FOR ( Cil_2_Gar_2_Ava == TRUE )
            WAIT FOR ( Cil_2_Gar_3_Ava == TRUE )
            WAIT FOR ( Cil_2_Gar_4_Ava == TRUE )
            WAIT FOR ( Cil_2_Gar_5_Ava == TRUE )
            WAIT FOR ( Cil_2_Gar_6_Ava == TRUE )

         CASE 171
            Abre_Gar_Triplo_Lado_A = TRUE
            Fecha_Gar_Triplo_Lado_A = FALSE

            Abre_Gar_Triplo_Lado_B = TRUE
            Fecha_Gar_Triplo_Lado_B = FALSE

            Abre_Comp_Indiv_Gar_1 = TRUE
            Fecha_Comp_Indiv_Gar_1 = FALSE

            Abre_Comp_Indiv_Gar_3 = FALSE
            Fecha_Comp_Indiv_Gar_3 = TRUE

            Abre_Comp_Indiv_Gar_4 = FALSE
            Fecha_Comp_Indiv_Gar_4 = TRUE

            Abre_Comp_Indiv_Gar_6 = FALSE
            Fecha_Comp_Indiv_Gar_6 = TRUE

            Ava_Cil_1_Gar_1 = TRUE
            Rec_Cil_1_Gar_1 = FALSE

            Ava_Cil_1_Gar_2 = TRUE
            Rec_Cil_1_Gar_2 = FALSE

            Ava_Cil_1_Gar_3 = TRUE
            Rec_Cil_1_Gar_3 = FALSE

            Ava_Cil_1_Gar_4 = TRUE
            Rec_Cil_1_Gar_4 = FALSE

            Ava_Cil_1_Gar_5 = TRUE
            Rec_Cil_1_Gar_5 = FALSE

            Ava_Cil_1_Gar_6 = TRUE
            Rec_Cil_1_Gar_6 = FALSE

            Ava_Cil_2_Gar_1 = TRUE
            Rec_Cil_2_Gar_1 = FALSE

            Ava_Cil_2_Gar_2 = TRUE
            Rec_Cil_2_Gar_2 = FALSE

            Ava_Cil_2_Gar_3 = TRUE
            Rec_Cil_2_Gar_3 = FALSE

            Ava_Cil_2_Gar_4 = TRUE
            Rec_Cil_2_Gar_4 = FALSE

            Ava_Cil_2_Gar_5 = TRUE
            Rec_Cil_2_Gar_5 = FALSE

            Ava_Cil_2_Gar_6 = TRUE
            Rec_Cil_2_Gar_6 = FALSE

            WAIT FOR ( Cil_Comp_Triplo_A_Ava == TRUE )
            WAIT FOR ( Cil_Comp_Triplo_A_Rec == FALSE )
            WAIT FOR ( Cil_Comp_Triplo_B_Ava == TRUE )
            WAIT FOR ( Cil_Comp_Triplo_B_Rec == FALSE )
            WAIT FOR ( Cil_Comp_Indiv_Gr_1_Aber == TRUE )
            WAIT FOR ( Cil_Comp_Indiv_Gr_1_Fech == FALSE )
            WAIT FOR ( Cil_Comp_Indiv_Gr_3_Aber == FALSE )
            WAIT FOR ( Cil_Comp_Indiv_Gr_3_Fech == TRUE )
            WAIT FOR ( Cil_Comp_Indiv_Gr_4_Aber == FALSE )
            WAIT FOR ( Cil_Comp_Indiv_Gr_4_Fech == TRUE )
            WAIT FOR ( Cil_Comp_Indiv_Gr_6_Aber == FALSE )
            WAIT FOR ( Cil_Comp_Indiv_Gr_6_Fech == TRUE )
            WAIT FOR ( Cil_1_Gar_1_Ava == TRUE )
            WAIT FOR ( Cil_1_Gar_2_Ava == TRUE )
            WAIT FOR ( Cil_1_Gar_3_Ava == TRUE )
            WAIT FOR ( Cil_1_Gar_4_Ava == TRUE )
            WAIT FOR ( Cil_1_Gar_5_Ava == TRUE )
            WAIT FOR ( Cil_1_Gar_6_Ava == TRUE )
            WAIT FOR ( Cil_2_Gar_1_Ava == TRUE )
            WAIT FOR ( Cil_2_Gar_2_Ava == TRUE )
            WAIT FOR ( Cil_2_Gar_3_Ava == TRUE )
            WAIT FOR ( Cil_2_Gar_4_Ava == TRUE )
            WAIT FOR ( Cil_2_Gar_5_Ava == TRUE )
            WAIT FOR ( Cil_2_Gar_6_Ava == TRUE )

         CASE 172
            Abre_Gar_Triplo_Lado_A = TRUE
            Fecha_Gar_Triplo_Lado_A = FALSE

            Abre_Gar_Triplo_Lado_B = TRUE
            Fecha_Gar_Triplo_Lado_B = FALSE

            Abre_Comp_Indiv_Gar_1 = TRUE
            Fecha_Comp_Indiv_Gar_1 = FALSE

            Abre_Comp_Indiv_Gar_3 = FALSE
            Fecha_Comp_Indiv_Gar_3 = TRUE

            Abre_Comp_Indiv_Gar_4 = FALSE
            Fecha_Comp_Indiv_Gar_4 = TRUE

            Abre_Comp_Indiv_Gar_6 = TRUE
            Fecha_Comp_Indiv_Gar_6 = FALSE

            Ava_Cil_1_Gar_1 = TRUE
            Rec_Cil_1_Gar_1 = FALSE

            Ava_Cil_1_Gar_2 = TRUE
            Rec_Cil_1_Gar_2 = FALSE

            Ava_Cil_1_Gar_3 = TRUE
            Rec_Cil_1_Gar_3 = FALSE

            Ava_Cil_1_Gar_4 = TRUE
            Rec_Cil_1_Gar_4 = FALSE

            Ava_Cil_1_Gar_5 = TRUE
            Rec_Cil_1_Gar_5 = FALSE

            Ava_Cil_1_Gar_6 = TRUE
            Rec_Cil_1_Gar_6 = FALSE

            Ava_Cil_2_Gar_1 = TRUE
            Rec_Cil_2_Gar_1 = FALSE

            Ava_Cil_2_Gar_2 = TRUE
            Rec_Cil_2_Gar_2 = FALSE

            Ava_Cil_2_Gar_3 = TRUE
            Rec_Cil_2_Gar_3 = FALSE

            Ava_Cil_2_Gar_4 = TRUE
            Rec_Cil_2_Gar_4 = FALSE

            Ava_Cil_2_Gar_5 = TRUE
            Rec_Cil_2_Gar_5 = FALSE

            Ava_Cil_2_Gar_6 = TRUE
            Rec_Cil_2_Gar_6 = FALSE

            WAIT FOR ( Cil_Comp_Triplo_A_Ava == FALSE )
            WAIT FOR ( Cil_Comp_Triplo_A_Rec == TRUE )
            WAIT FOR ( Cil_Comp_Triplo_B_Ava == FALSE )
            WAIT FOR ( Cil_Comp_Triplo_B_Rec == TRUE )
            WAIT FOR ( Cil_Comp_Indiv_Gr_1_Aber == TRUE )
            WAIT FOR ( Cil_Comp_Indiv_Gr_1_Fech == FALSE )
            WAIT FOR ( Cil_Comp_Indiv_Gr_3_Aber == FALSE )
            WAIT FOR ( Cil_Comp_Indiv_Gr_3_Fech == TRUE )
            WAIT FOR ( Cil_Comp_Indiv_Gr_4_Aber == FALSE )
            WAIT FOR ( Cil_Comp_Indiv_Gr_4_Fech == TRUE )
            WAIT FOR ( Cil_Comp_Indiv_Gr_6_Aber == TRUE )
            WAIT FOR ( Cil_Comp_Indiv_Gr_6_Fech == FALSE )
            WAIT FOR ( Cil_1_Gar_1_Ava == TRUE )
            WAIT FOR ( Cil_1_Gar_2_Ava == TRUE )
            WAIT FOR ( Cil_1_Gar_3_Ava == TRUE )
            WAIT FOR ( Cil_1_Gar_4_Ava == TRUE )
            WAIT FOR ( Cil_1_Gar_5_Ava == TRUE )
            WAIT FOR ( Cil_1_Gar_6_Ava == TRUE )
            WAIT FOR ( Cil_2_Gar_1_Ava == TRUE )
            WAIT FOR ( Cil_2_Gar_2_Ava == TRUE )
            WAIT FOR ( Cil_2_Gar_3_Ava == TRUE )
            WAIT FOR ( Cil_2_Gar_4_Ava == TRUE )
            WAIT FOR ( Cil_2_Gar_5_Ava == TRUE )
            WAIT FOR ( Cil_2_Gar_6_Ava == TRUE )

         CASE 173
            Abre_Gar_Triplo_Lado_A = TRUE
            Fecha_Gar_Triplo_Lado_A = FALSE

            Abre_Gar_Triplo_Lado_B = TRUE
            Fecha_Gar_Triplo_Lado_B = FALSE

            Abre_Comp_Indiv_Gar_1 = TRUE
            Fecha_Comp_Indiv_Gar_1 = FALSE

            Abre_Comp_Indiv_Gar_3 = FALSE
            Fecha_Comp_Indiv_Gar_3 = TRUE

            Abre_Comp_Indiv_Gar_4 = FALSE
            Fecha_Comp_Indiv_Gar_4 = TRUE

            Abre_Comp_Indiv_Gar_6 = TRUE
            Fecha_Comp_Indiv_Gar_6 = FALSE

            Ava_Cil_1_Gar_1 = TRUE
            Rec_Cil_1_Gar_1 = FALSE

            Ava_Cil_1_Gar_2 = TRUE
            Rec_Cil_1_Gar_2 = FALSE

            Ava_Cil_1_Gar_3 = TRUE
            Rec_Cil_1_Gar_3 = FALSE

            Ava_Cil_1_Gar_4 = TRUE
            Rec_Cil_1_Gar_4 = FALSE

            Ava_Cil_1_Gar_5 = TRUE
            Rec_Cil_1_Gar_5 = FALSE

            Ava_Cil_1_Gar_6 = TRUE
            Rec_Cil_1_Gar_6 = FALSE

            Ava_Cil_2_Gar_1 = TRUE
            Rec_Cil_2_Gar_1 = FALSE

            Ava_Cil_2_Gar_2 = TRUE
            Rec_Cil_2_Gar_2 = FALSE

            Ava_Cil_2_Gar_3 = TRUE
            Rec_Cil_2_Gar_3 = FALSE

            Ava_Cil_2_Gar_4 = TRUE
            Rec_Cil_2_Gar_4 = FALSE

            Ava_Cil_2_Gar_5 = TRUE
            Rec_Cil_2_Gar_5 = FALSE

            Ava_Cil_2_Gar_6 = TRUE
            Rec_Cil_2_Gar_6 = FALSE

            WAIT FOR ( Cil_Comp_Triplo_A_Ava == FALSE )
            WAIT FOR ( Cil_Comp_Triplo_A_Rec == TRUE )
            WAIT FOR ( Cil_Comp_Triplo_B_Ava == FALSE )
            WAIT FOR ( Cil_Comp_Triplo_B_Rec == TRUE )
            WAIT FOR ( Cil_Comp_Indiv_Gr_1_Aber == TRUE )
            WAIT FOR ( Cil_Comp_Indiv_Gr_1_Fech == FALSE )
            WAIT FOR ( Cil_Comp_Indiv_Gr_3_Aber == FALSE )
            WAIT FOR ( Cil_Comp_Indiv_Gr_3_Fech == TRUE )
            WAIT FOR ( Cil_Comp_Indiv_Gr_4_Aber == FALSE )
            WAIT FOR ( Cil_Comp_Indiv_Gr_4_Fech == TRUE )
            WAIT FOR ( Cil_Comp_Indiv_Gr_6_Aber == TRUE )
            WAIT FOR ( Cil_Comp_Indiv_Gr_6_Fech == FALSE )
            WAIT FOR ( Cil_1_Gar_1_Ava == TRUE )
            WAIT FOR ( Cil_1_Gar_2_Ava == TRUE )
            WAIT FOR ( Cil_1_Gar_3_Ava == TRUE )
            WAIT FOR ( Cil_1_Gar_4_Ava == TRUE )
            WAIT FOR ( Cil_1_Gar_5_Ava == TRUE )
            WAIT FOR ( Cil_1_Gar_6_Ava == TRUE )
            WAIT FOR ( Cil_2_Gar_1_Ava == TRUE )
            WAIT FOR ( Cil_2_Gar_2_Ava == TRUE )
            WAIT FOR ( Cil_2_Gar_3_Ava == TRUE )
            WAIT FOR ( Cil_2_Gar_4_Ava == TRUE )
            WAIT FOR ( Cil_2_Gar_5_Ava == TRUE )
            WAIT FOR ( Cil_2_Gar_6_Ava == TRUE )

         CASE 71
            Abre_Gar_Triplo_Lado_A = TRUE
            Fecha_Gar_Triplo_Lado_A = FALSE

            Abre_Gar_Triplo_Lado_B = TRUE
            Fecha_Gar_Triplo_Lado_B = FALSE

            Abre_Comp_Indiv_Gar_1 = FALSE
            Fecha_Comp_Indiv_Gar_1 = TRUE

            Abre_Comp_Indiv_Gar_3 = TRUE
            Fecha_Comp_Indiv_Gar_3 = FALSE

            Abre_Comp_Indiv_Gar_4 = TRUE
            Fecha_Comp_Indiv_Gar_4 = FALSE

            Abre_Comp_Indiv_Gar_6 = FALSE
            Fecha_Comp_Indiv_Gar_6 = TRUE

            Ava_Cil_1_Gar_1 = TRUE
            Rec_Cil_1_Gar_1 = FALSE

            Ava_Cil_1_Gar_2 = TRUE
            Rec_Cil_1_Gar_2 = FALSE

            Ava_Cil_1_Gar_3 = TRUE
            Rec_Cil_1_Gar_3 = FALSE

            Ava_Cil_1_Gar_4 = TRUE
            Rec_Cil_1_Gar_4 = FALSE

            Ava_Cil_1_Gar_5 = TRUE
            Rec_Cil_1_Gar_5 = FALSE

            Ava_Cil_1_Gar_6 = TRUE
            Rec_Cil_1_Gar_6 = FALSE

            Ava_Cil_2_Gar_1 = TRUE
            Rec_Cil_2_Gar_1 = FALSE

            Ava_Cil_2_Gar_2 = TRUE
            Rec_Cil_2_Gar_2 = FALSE

            Ava_Cil_2_Gar_3 = TRUE
            Rec_Cil_2_Gar_3 = FALSE

            Ava_Cil_2_Gar_4 = TRUE
            Rec_Cil_2_Gar_4 = FALSE

            Ava_Cil_2_Gar_5 = TRUE
            Rec_Cil_2_Gar_5 = FALSE

            Ava_Cil_2_Gar_6 = TRUE
            Rec_Cil_2_Gar_6 = FALSE

            WAIT FOR ( Cil_Comp_Triplo_A_Ava == FALSE )
            WAIT FOR ( Cil_Comp_Triplo_A_Rec == TRUE )
            WAIT FOR ( Cil_Comp_Triplo_B_Ava == FALSE )
            WAIT FOR ( Cil_Comp_Triplo_B_Rec == TRUE )
            WAIT FOR ( Cil_Comp_Indiv_Gr_1_Aber == FALSE )
            WAIT FOR ( Cil_Comp_Indiv_Gr_1_Fech == TRUE )
            WAIT FOR ( Cil_Comp_Indiv_Gr_3_Aber == TRUE )
            WAIT FOR ( Cil_Comp_Indiv_Gr_3_Fech == FALSE )
            WAIT FOR ( Cil_Comp_Indiv_Gr_4_Aber == TRUE )
            WAIT FOR ( Cil_Comp_Indiv_Gr_4_Fech == FALSE )
            WAIT FOR ( Cil_Comp_Indiv_Gr_6_Aber == FALSE )
            WAIT FOR ( Cil_Comp_Indiv_Gr_6_Fech == TRUE )
            WAIT FOR ( Cil_1_Gar_1_Ava == TRUE )
            WAIT FOR ( Cil_1_Gar_2_Ava == TRUE )
            WAIT FOR ( Cil_1_Gar_3_Ava == TRUE )
            WAIT FOR ( Cil_1_Gar_4_Ava == TRUE )
            WAIT FOR ( Cil_1_Gar_5_Ava == TRUE )
            WAIT FOR ( Cil_1_Gar_6_Ava == TRUE )
            WAIT FOR ( Cil_2_Gar_1_Ava == TRUE )
            WAIT FOR ( Cil_2_Gar_2_Ava == TRUE )
            WAIT FOR ( Cil_2_Gar_3_Ava == TRUE )
            WAIT FOR ( Cil_2_Gar_4_Ava == TRUE )
            WAIT FOR ( Cil_2_Gar_5_Ava == TRUE )
            WAIT FOR ( Cil_2_Gar_6_Ava == TRUE )

         CASE 72
            Abre_Gar_Triplo_Lado_A = TRUE
            Fecha_Gar_Triplo_Lado_A = FALSE

            Abre_Gar_Triplo_Lado_B = TRUE
            Fecha_Gar_Triplo_Lado_B = FALSE

            Abre_Comp_Indiv_Gar_1 = TRUE
            Fecha_Comp_Indiv_Gar_1 = FALSE

            Abre_Comp_Indiv_Gar_3 = FALSE
            Fecha_Comp_Indiv_Gar_3 = TRUE

            Abre_Comp_Indiv_Gar_4 = TRUE
            Fecha_Comp_Indiv_Gar_4 = FALSE

            Abre_Comp_Indiv_Gar_6 = FALSE
            Fecha_Comp_Indiv_Gar_6 = TRUE

            Ava_Cil_1_Gar_1 = TRUE
            Rec_Cil_1_Gar_1 = FALSE

            Ava_Cil_1_Gar_2 = TRUE
            Rec_Cil_1_Gar_2 = FALSE

            Ava_Cil_1_Gar_3 = TRUE
            Rec_Cil_1_Gar_3 = FALSE

            Ava_Cil_1_Gar_4 = TRUE
            Rec_Cil_1_Gar_4 = FALSE

            Ava_Cil_1_Gar_5 = TRUE
            Rec_Cil_1_Gar_5 = FALSE

            Ava_Cil_1_Gar_6 = TRUE
            Rec_Cil_1_Gar_6 = FALSE

            Ava_Cil_2_Gar_1 = TRUE
            Rec_Cil_2_Gar_1 = FALSE

            Ava_Cil_2_Gar_2 = TRUE
            Rec_Cil_2_Gar_2 = FALSE

            Ava_Cil_2_Gar_3 = TRUE
            Rec_Cil_2_Gar_3 = FALSE

            Ava_Cil_2_Gar_4 = TRUE
            Rec_Cil_2_Gar_4 = FALSE

            Ava_Cil_2_Gar_5 = TRUE
            Rec_Cil_2_Gar_5 = FALSE

            Ava_Cil_2_Gar_6 = TRUE
            Rec_Cil_2_Gar_6 = FALSE

            WAIT FOR ( Cil_Comp_Triplo_A_Ava == FALSE )
            WAIT FOR ( Cil_Comp_Triplo_A_Rec == TRUE )
            WAIT FOR ( Cil_Comp_Triplo_B_Ava == FALSE )
            WAIT FOR ( Cil_Comp_Triplo_B_Rec == TRUE )
            WAIT FOR ( Cil_Comp_Indiv_Gr_1_Aber == TRUE )
            WAIT FOR ( Cil_Comp_Indiv_Gr_1_Fech == FALSE )
            WAIT FOR ( Cil_Comp_Indiv_Gr_3_Aber == FALSE )
            WAIT FOR ( Cil_Comp_Indiv_Gr_3_Fech == TRUE )
            WAIT FOR ( Cil_Comp_Indiv_Gr_4_Aber == TRUE )
            WAIT FOR ( Cil_Comp_Indiv_Gr_4_Fech == FALSE )
            WAIT FOR ( Cil_Comp_Indiv_Gr_6_Aber == FALSE )
            WAIT FOR ( Cil_Comp_Indiv_Gr_6_Fech == TRUE )
            WAIT FOR ( Cil_1_Gar_1_Ava == TRUE )
            WAIT FOR ( Cil_1_Gar_2_Ava == TRUE )
            WAIT FOR ( Cil_1_Gar_3_Ava == TRUE )
            WAIT FOR ( Cil_1_Gar_4_Ava == TRUE )
            WAIT FOR ( Cil_1_Gar_5_Ava == TRUE )
            WAIT FOR ( Cil_1_Gar_6_Ava == TRUE )
            WAIT FOR ( Cil_2_Gar_1_Ava == TRUE )
            WAIT FOR ( Cil_2_Gar_2_Ava == TRUE )
            WAIT FOR ( Cil_2_Gar_3_Ava == TRUE )
            WAIT FOR ( Cil_2_Gar_4_Ava == TRUE )
            WAIT FOR ( Cil_2_Gar_5_Ava == TRUE )
            WAIT FOR ( Cil_2_Gar_6_Ava == TRUE )

         CASE 73
            Abre_Gar_Triplo_Lado_A = TRUE
            Fecha_Gar_Triplo_Lado_A = FALSE

            Abre_Gar_Triplo_Lado_B = TRUE
            Fecha_Gar_Triplo_Lado_B = FALSE

            Abre_Comp_Indiv_Gar_1 = TRUE
            Fecha_Comp_Indiv_Gar_1 = FALSE

            Abre_Comp_Indiv_Gar_3 = TRUE
            Fecha_Comp_Indiv_Gar_3 = FALSE

            Abre_Comp_Indiv_Gar_4 = TRUE
            Fecha_Comp_Indiv_Gar_4 = FALSE

            Abre_Comp_Indiv_Gar_6 = TRUE
            Fecha_Comp_Indiv_Gar_6 = FALSE

            Ava_Cil_1_Gar_1 = TRUE
            Rec_Cil_1_Gar_1 = FALSE

            Ava_Cil_1_Gar_2 = TRUE
            Rec_Cil_1_Gar_2 = FALSE

            Ava_Cil_1_Gar_3 = TRUE
            Rec_Cil_1_Gar_3 = FALSE

            Ava_Cil_1_Gar_4 = TRUE
            Rec_Cil_1_Gar_4 = FALSE

            Ava_Cil_1_Gar_5 = TRUE
            Rec_Cil_1_Gar_5 = FALSE

            Ava_Cil_1_Gar_6 = TRUE
            Rec_Cil_1_Gar_6 = FALSE

            Ava_Cil_2_Gar_1 = TRUE
            Rec_Cil_2_Gar_1 = FALSE

            Ava_Cil_2_Gar_2 = TRUE
            Rec_Cil_2_Gar_2 = FALSE

            Ava_Cil_2_Gar_3 = TRUE
            Rec_Cil_2_Gar_3 = FALSE

            Ava_Cil_2_Gar_4 = TRUE
            Rec_Cil_2_Gar_4 = FALSE

            Ava_Cil_2_Gar_5 = TRUE
            Rec_Cil_2_Gar_5 = FALSE

            Ava_Cil_2_Gar_6 = TRUE
            Rec_Cil_2_Gar_6 = FALSE

            WAIT FOR ( Cil_Comp_Triplo_A_Ava == FALSE )
            WAIT FOR ( Cil_Comp_Triplo_A_Rec == TRUE )
            WAIT FOR ( Cil_Comp_Triplo_B_Ava == FALSE )
            WAIT FOR ( Cil_Comp_Triplo_B_Rec == TRUE )
            WAIT FOR ( Cil_Comp_Indiv_Gr_1_Aber == TRUE )
            WAIT FOR ( Cil_Comp_Indiv_Gr_1_Fech == FALSE )
            WAIT FOR ( Cil_Comp_Indiv_Gr_3_Aber == TRUE )
            WAIT FOR ( Cil_Comp_Indiv_Gr_3_Fech == FALSE )
            WAIT FOR ( Cil_Comp_Indiv_Gr_4_Aber == TRUE )
            WAIT FOR ( Cil_Comp_Indiv_Gr_4_Fech == FALSE )
            WAIT FOR ( Cil_Comp_Indiv_Gr_6_Aber == TRUE )
            WAIT FOR ( Cil_Comp_Indiv_Gr_6_Fech == FALSE )
            WAIT FOR ( Cil_1_Gar_1_Ava == TRUE )
            WAIT FOR ( Cil_1_Gar_2_Ava == TRUE )
            WAIT FOR ( Cil_1_Gar_3_Ava == TRUE )
            WAIT FOR ( Cil_1_Gar_4_Ava == TRUE )
            WAIT FOR ( Cil_1_Gar_5_Ava == TRUE )
            WAIT FOR ( Cil_1_Gar_6_Ava == TRUE )
            WAIT FOR ( Cil_2_Gar_1_Ava == TRUE )
            WAIT FOR ( Cil_2_Gar_2_Ava == TRUE )
            WAIT FOR ( Cil_2_Gar_3_Ava == TRUE )
            WAIT FOR ( Cil_2_Gar_4_Ava == TRUE )
            WAIT FOR ( Cil_2_Gar_5_Ava == TRUE )
            WAIT FOR ( Cil_2_Gar_6_Ava == TRUE )

         CASE 51
            Abre_Gar_Triplo_Lado_A = TRUE
            Fecha_Gar_Triplo_Lado_A = FALSE

            Abre_Gar_Triplo_Lado_B = TRUE
            Fecha_Gar_Triplo_Lado_B = FALSE

            Abre_Comp_Indiv_Gar_1 = TRUE
            Fecha_Comp_Indiv_Gar_1 = FALSE

            Abre_Comp_Indiv_Gar_3 = TRUE
            Fecha_Comp_Indiv_Gar_3 = FALSE

            Abre_Comp_Indiv_Gar_4 = TRUE
            Fecha_Comp_Indiv_Gar_4 = FALSE

            Abre_Comp_Indiv_Gar_6 = TRUE
            Fecha_Comp_Indiv_Gar_6 = FALSE

            Ava_Cil_1_Gar_1 = TRUE
            Rec_Cil_1_Gar_1 = FALSE

            Ava_Cil_1_Gar_2 = TRUE
            Rec_Cil_1_Gar_2 = FALSE

            Ava_Cil_1_Gar_3 = TRUE
            Rec_Cil_1_Gar_3 = FALSE

            Ava_Cil_1_Gar_4 = TRUE
            Rec_Cil_1_Gar_4 = FALSE

            Ava_Cil_1_Gar_5 = TRUE
            Rec_Cil_1_Gar_5 = FALSE

            Ava_Cil_1_Gar_6 = TRUE
            Rec_Cil_1_Gar_6 = FALSE

            Ava_Cil_2_Gar_1 = TRUE
            Rec_Cil_2_Gar_1 = FALSE

            Ava_Cil_2_Gar_2 = TRUE
            Rec_Cil_2_Gar_2 = FALSE

            Ava_Cil_2_Gar_3 = TRUE
            Rec_Cil_2_Gar_3 = FALSE

            Ava_Cil_2_Gar_4 = TRUE
            Rec_Cil_2_Gar_4 = FALSE

            Ava_Cil_2_Gar_5 = TRUE
            Rec_Cil_2_Gar_5 = FALSE

            Ava_Cil_2_Gar_6 = TRUE
            Rec_Cil_2_Gar_6 = FALSE

            WAIT FOR ( Cil_Comp_Triplo_A_Ava == FALSE )
            WAIT FOR ( Cil_Comp_Triplo_A_Rec == TRUE )
            WAIT FOR ( Cil_Comp_Triplo_B_Ava == FALSE )
            WAIT FOR ( Cil_Comp_Triplo_B_Rec == TRUE )
            WAIT FOR ( Cil_Comp_Indiv_Gr_1_Aber == TRUE )
            WAIT FOR ( Cil_Comp_Indiv_Gr_1_Fech == FALSE )
            WAIT FOR ( Cil_Comp_Indiv_Gr_3_Aber == TRUE )
            WAIT FOR ( Cil_Comp_Indiv_Gr_3_Fech == FALSE )
            WAIT FOR ( Cil_Comp_Indiv_Gr_4_Aber == TRUE )
            WAIT FOR ( Cil_Comp_Indiv_Gr_4_Fech == FALSE )
            WAIT FOR ( Cil_Comp_Indiv_Gr_6_Aber == TRUE )
            WAIT FOR ( Cil_Comp_Indiv_Gr_6_Fech == FALSE )
            WAIT FOR ( Cil_1_Gar_1_Ava == TRUE )
            WAIT FOR ( Cil_1_Gar_2_Ava == TRUE )
            WAIT FOR ( Cil_1_Gar_3_Ava == TRUE )
            WAIT FOR ( Cil_1_Gar_4_Ava == TRUE )
            WAIT FOR ( Cil_1_Gar_5_Ava == TRUE )
            WAIT FOR ( Cil_1_Gar_6_Ava == TRUE )
            WAIT FOR ( Cil_2_Gar_1_Ava == TRUE )
            WAIT FOR ( Cil_2_Gar_2_Ava == TRUE )
            WAIT FOR ( Cil_2_Gar_3_Ava == TRUE )
            WAIT FOR ( Cil_2_Gar_4_Ava == TRUE )
            WAIT FOR ( Cil_2_Gar_5_Ava == TRUE )
            WAIT FOR ( Cil_2_Gar_6_Ava == TRUE )

         CASE 131
            Abre_Gar_Triplo_Lado_A = TRUE
            Fecha_Gar_Triplo_Lado_A = FALSE

            Abre_Gar_Triplo_Lado_B = TRUE
            Fecha_Gar_Triplo_Lado_B = FALSE

            Abre_Comp_Indiv_Gar_1 = TRUE
            Fecha_Comp_Indiv_Gar_1 = FALSE

            Abre_Comp_Indiv_Gar_3 = TRUE
            Fecha_Comp_Indiv_Gar_3 = FALSE

            Abre_Comp_Indiv_Gar_4 = TRUE
            Fecha_Comp_Indiv_Gar_4 = FALSE

            Abre_Comp_Indiv_Gar_6 = TRUE
            Fecha_Comp_Indiv_Gar_6 = FALSE

            Ava_Cil_1_Gar_1 = TRUE
            Rec_Cil_1_Gar_1 = FALSE

            Ava_Cil_1_Gar_2 = TRUE
            Rec_Cil_1_Gar_2 = FALSE

            Ava_Cil_1_Gar_3 = TRUE
            Rec_Cil_1_Gar_3 = FALSE

            Ava_Cil_1_Gar_4 = TRUE
            Rec_Cil_1_Gar_4 = FALSE

            Ava_Cil_1_Gar_5 = TRUE
            Rec_Cil_1_Gar_5 = FALSE

            Ava_Cil_1_Gar_6 = TRUE
            Rec_Cil_1_Gar_6 = FALSE

            Ava_Cil_2_Gar_1 = TRUE
            Rec_Cil_2_Gar_1 = FALSE

            Ava_Cil_2_Gar_2 = TRUE
            Rec_Cil_2_Gar_2 = FALSE

            Ava_Cil_2_Gar_3 = TRUE
            Rec_Cil_2_Gar_3 = FALSE

            Ava_Cil_2_Gar_4 = TRUE
            Rec_Cil_2_Gar_4 = FALSE

            Ava_Cil_2_Gar_5 = TRUE
            Rec_Cil_2_Gar_5 = FALSE

            Ava_Cil_2_Gar_6 = TRUE
            Rec_Cil_2_Gar_6 = FALSE

            WAIT FOR ( Cil_Comp_Triplo_A_Ava == FALSE )
            WAIT FOR ( Cil_Comp_Triplo_A_Rec == TRUE )
            WAIT FOR ( Cil_Comp_Triplo_B_Ava == FALSE )
            WAIT FOR ( Cil_Comp_Triplo_B_Rec == TRUE )
            WAIT FOR ( Cil_Comp_Indiv_Gr_1_Aber == TRUE )
            WAIT FOR ( Cil_Comp_Indiv_Gr_1_Fech == FALSE )
            WAIT FOR ( Cil_Comp_Indiv_Gr_3_Aber == TRUE )
            WAIT FOR ( Cil_Comp_Indiv_Gr_3_Fech == FALSE )
            WAIT FOR ( Cil_Comp_Indiv_Gr_4_Aber == TRUE )
            WAIT FOR ( Cil_Comp_Indiv_Gr_4_Fech == FALSE )
            WAIT FOR ( Cil_Comp_Indiv_Gr_6_Aber == TRUE )
            WAIT FOR ( Cil_Comp_Indiv_Gr_6_Fech == FALSE )
            WAIT FOR ( Cil_1_Gar_1_Ava == TRUE )
            WAIT FOR ( Cil_1_Gar_2_Ava == TRUE )
            WAIT FOR ( Cil_1_Gar_3_Ava == TRUE )
            WAIT FOR ( Cil_1_Gar_4_Ava == TRUE )
            WAIT FOR ( Cil_1_Gar_5_Ava == TRUE )
            WAIT FOR ( Cil_1_Gar_6_Ava == TRUE )
            WAIT FOR ( Cil_2_Gar_1_Ava == TRUE )
            WAIT FOR ( Cil_2_Gar_2_Ava == TRUE )
            WAIT FOR ( Cil_2_Gar_3_Ava == TRUE )
            WAIT FOR ( Cil_2_Gar_4_Ava == TRUE )
            WAIT FOR ( Cil_2_Gar_5_Ava == TRUE )
            WAIT FOR ( Cil_2_Gar_6_Ava == TRUE )
         CASE 181
            Abre_Gar_Triplo_Lado_A = TRUE
            Fecha_Gar_Triplo_Lado_A = FALSE

            Abre_Gar_Triplo_Lado_B = TRUE
            Fecha_Gar_Triplo_Lado_B = FALSE

            Abre_Comp_Indiv_Gar_1 = FALSE
            Fecha_Comp_Indiv_Gar_1 = TRUE

            Abre_Comp_Indiv_Gar_3 = FALSE
            Fecha_Comp_Indiv_Gar_3 = TRUE

            Abre_Comp_Indiv_Gar_4 = FALSE
            Fecha_Comp_Indiv_Gar_4 = TRUE

            Abre_Comp_Indiv_Gar_6 = FALSE
            Fecha_Comp_Indiv_Gar_6 = TRUE

            Ava_Cil_1_Gar_1 = TRUE
            Rec_Cil_1_Gar_1 = FALSE

            Ava_Cil_1_Gar_2 = TRUE
            Rec_Cil_1_Gar_2 = FALSE

            Ava_Cil_1_Gar_3 = TRUE
            Rec_Cil_1_Gar_3 = FALSE

            Ava_Cil_1_Gar_4 = TRUE
            Rec_Cil_1_Gar_4 = FALSE

            Ava_Cil_1_Gar_5 = TRUE
            Rec_Cil_1_Gar_5 = FALSE

            Ava_Cil_1_Gar_6 = TRUE
            Rec_Cil_1_Gar_6 = FALSE

            Ava_Cil_2_Gar_1 = TRUE
            Rec_Cil_2_Gar_1 = FALSE

            Ava_Cil_2_Gar_2 = TRUE
            Rec_Cil_2_Gar_2 = FALSE

            Ava_Cil_2_Gar_3 = TRUE
            Rec_Cil_2_Gar_3 = FALSE

            Ava_Cil_2_Gar_4 = TRUE
            Rec_Cil_2_Gar_4 = FALSE

            Ava_Cil_2_Gar_5 = TRUE
            Rec_Cil_2_Gar_5 = FALSE

            Ava_Cil_2_Gar_6 = TRUE
            Rec_Cil_2_Gar_6 = FALSE

            WAIT FOR ( Cil_Comp_Triplo_A_Ava == FALSE )
            WAIT FOR ( Cil_Comp_Triplo_A_Rec == TRUE )
            WAIT FOR ( Cil_Comp_Triplo_B_Ava == TRUE )
            WAIT FOR ( Cil_Comp_Triplo_B_Rec == FALSE )
            WAIT FOR ( Cil_Comp_Indiv_Gr_1_Aber == FALSE )
            WAIT FOR ( Cil_Comp_Indiv_Gr_1_Fech == TRUE )
            WAIT FOR ( Cil_Comp_Indiv_Gr_3_Aber == FALSE )
            WAIT FOR ( Cil_Comp_Indiv_Gr_3_Fech == TRUE )
            WAIT FOR ( Cil_Comp_Indiv_Gr_4_Aber == FALSE )
            WAIT FOR ( Cil_Comp_Indiv_Gr_4_Fech == TRUE )
            WAIT FOR ( Cil_Comp_Indiv_Gr_6_Aber == FALSE )
            WAIT FOR ( Cil_Comp_Indiv_Gr_6_Fech == TRUE )
            WAIT FOR ( Cil_1_Gar_1_Ava == TRUE )
            WAIT FOR ( Cil_1_Gar_2_Ava == TRUE )
            WAIT FOR ( Cil_1_Gar_3_Ava == TRUE )
            WAIT FOR ( Cil_1_Gar_4_Ava == TRUE )
            WAIT FOR ( Cil_1_Gar_5_Ava == TRUE )
            WAIT FOR ( Cil_1_Gar_6_Ava == TRUE )
            WAIT FOR ( Cil_2_Gar_1_Ava == TRUE )
            WAIT FOR ( Cil_2_Gar_2_Ava == TRUE )
            WAIT FOR ( Cil_2_Gar_3_Ava == TRUE )
            WAIT FOR ( Cil_2_Gar_4_Ava == TRUE )
            WAIT FOR ( Cil_2_Gar_5_Ava == TRUE )
            WAIT FOR ( Cil_2_Gar_6_Ava == TRUE )

      ENDSWITCH


END

Global Def ConfGarra_nowait()

      SWITCH ConfGarraOp
         CASE 11
            Abre_Gar_Triplo_Lado_A = TRUE
            Fecha_Gar_Triplo_Lado_A = FALSE

            Abre_Gar_Triplo_Lado_B = TRUE
            Fecha_Gar_Triplo_Lado_B = FALSE

            Abre_Comp_Indiv_Gar_1 = FALSE
            Fecha_Comp_Indiv_Gar_1 = TRUE

            Abre_Comp_Indiv_Gar_3 = TRUE
            Fecha_Comp_Indiv_Gar_3 = FALSE

            Abre_Comp_Indiv_Gar_4 = FALSE
            Fecha_Comp_Indiv_Gar_4 = TRUE

            Abre_Comp_Indiv_Gar_6 = TRUE
            Fecha_Comp_Indiv_Gar_6 = FALSE

            Ava_Cil_2_Gar_1 = TRUE
            Rec_Cil_2_Gar_1 = FALSE

            Ava_Cil_2_Gar_2 = TRUE
            Rec_Cil_2_Gar_2 = FALSE

            Ava_Cil_2_Gar_3 = TRUE
            Rec_Cil_2_Gar_3 = FALSE

            Ava_Cil_2_Gar_4 = TRUE
            Rec_Cil_2_Gar_4 = FALSE

            Ava_Cil_2_Gar_5 = TRUE
            Rec_Cil_2_Gar_5 = FALSE

            Ava_Cil_2_Gar_6 = TRUE
            Rec_Cil_2_Gar_6 = FALSE

            Ava_Cil_1_Gar_1 = TRUE
            Rec_Cil_1_Gar_1 = FALSE

            Ava_Cil_1_Gar_2 = TRUE
            Rec_Cil_1_Gar_2 = FALSE

            Ava_Cil_1_Gar_3 = TRUE
            Rec_Cil_1_Gar_3 = FALSE

            Ava_Cil_1_Gar_4 = TRUE
            Rec_Cil_1_Gar_4 = FALSE

            Ava_Cil_1_Gar_5 = TRUE
            Rec_Cil_1_Gar_5 = FALSE

            Ava_Cil_1_Gar_6 = TRUE
            Rec_Cil_1_Gar_6 = FALSE

         CASE 21
            Abre_Gar_Triplo_Lado_A = TRUE
            Fecha_Gar_Triplo_Lado_A = FALSE

            Abre_Gar_Triplo_Lado_B = TRUE
            Fecha_Gar_Triplo_Lado_B = FALSE

            Abre_Comp_Indiv_Gar_1 = FALSE
            Fecha_Comp_Indiv_Gar_1 = TRUE

            Abre_Comp_Indiv_Gar_3 = FALSE
            Fecha_Comp_Indiv_Gar_3 = TRUE

            Abre_Comp_Indiv_Gar_4 = FALSE
            Fecha_Comp_Indiv_Gar_4 = TRUE

            Abre_Comp_Indiv_Gar_6 = FALSE
            Fecha_Comp_Indiv_Gar_6 = TRUE

            Ava_Cil_2_Gar_1 = TRUE
            Rec_Cil_2_Gar_1 = FALSE

            Ava_Cil_2_Gar_2 = TRUE
            Rec_Cil_2_Gar_2 = FALSE

            Ava_Cil_2_Gar_3 = TRUE
            Rec_Cil_2_Gar_3 = FALSE

            Ava_Cil_2_Gar_4 = TRUE
            Rec_Cil_2_Gar_4 = FALSE

            Ava_Cil_2_Gar_5 = TRUE
            Rec_Cil_2_Gar_5 = FALSE

            Ava_Cil_2_Gar_6 = TRUE
            Rec_Cil_2_Gar_6 = FALSE

            Ava_Cil_1_Gar_1 = TRUE
            Rec_Cil_1_Gar_1 = FALSE

            Ava_Cil_1_Gar_2 = TRUE
            Rec_Cil_1_Gar_2 = FALSE

            Ava_Cil_1_Gar_3 = TRUE
            Rec_Cil_1_Gar_3 = FALSE

            Ava_Cil_1_Gar_4 = TRUE
            Rec_Cil_1_Gar_4 = FALSE

            Ava_Cil_1_Gar_5 = TRUE
            Rec_Cil_1_Gar_5 = FALSE

            Ava_Cil_1_Gar_6 = TRUE
            Rec_Cil_1_Gar_6 = FALSE



         CASE 101
            Abre_Gar_Triplo_Lado_A = TRUE
            Fecha_Gar_Triplo_Lado_A = FALSE

            Abre_Gar_Triplo_Lado_B = TRUE
            Fecha_Gar_Triplo_Lado_B = FALSE

            Abre_Comp_Indiv_Gar_1 = TRUE
            Fecha_Comp_Indiv_Gar_1 = FALSE

            Abre_Comp_Indiv_Gar_3 = FALSE
            Fecha_Comp_Indiv_Gar_3 = TRUE

            Abre_Comp_Indiv_Gar_4 = FALSE
            Fecha_Comp_Indiv_Gar_4 = TRUE

            Abre_Comp_Indiv_Gar_6 = TRUE
            Fecha_Comp_Indiv_Gar_6 = FALSE

            Ava_Cil_2_Gar_1 = TRUE
            Rec_Cil_2_Gar_1 = FALSE

            Ava_Cil_2_Gar_2 = TRUE
            Rec_Cil_2_Gar_2 = FALSE

            Ava_Cil_2_Gar_3 = TRUE
            Rec_Cil_2_Gar_3 = FALSE

            Ava_Cil_2_Gar_4 = TRUE
            Rec_Cil_2_Gar_4 = FALSE

            Ava_Cil_2_Gar_5 = TRUE
            Rec_Cil_2_Gar_5 = FALSE

            Ava_Cil_2_Gar_6 = TRUE
            Rec_Cil_2_Gar_6 = FALSE

            Ava_Cil_1_Gar_1 = TRUE
            Rec_Cil_1_Gar_1 = FALSE

            Ava_Cil_1_Gar_2 = TRUE
            Rec_Cil_1_Gar_2 = FALSE

            Ava_Cil_1_Gar_3 = TRUE
            Rec_Cil_1_Gar_3 = FALSE

            Ava_Cil_1_Gar_4 = TRUE
            Rec_Cil_1_Gar_4 = FALSE

            Ava_Cil_1_Gar_5 = TRUE
            Rec_Cil_1_Gar_5 = FALSE

            Ava_Cil_1_Gar_6 = TRUE
            Rec_Cil_1_Gar_6 = FALSE

         CASE 102
            Abre_Gar_Triplo_Lado_A = TRUE
            Fecha_Gar_Triplo_Lado_A = FALSE

            Abre_Gar_Triplo_Lado_B = TRUE
            Fecha_Gar_Triplo_Lado_B = FALSE

            Abre_Comp_Indiv_Gar_1 = TRUE
            Fecha_Comp_Indiv_Gar_1 = FALSE

            Abre_Comp_Indiv_Gar_3 = FALSE
            Fecha_Comp_Indiv_Gar_3 = TRUE

            Abre_Comp_Indiv_Gar_4 = FALSE
            Fecha_Comp_Indiv_Gar_4 = TRUE

            Abre_Comp_Indiv_Gar_6 = TRUE
            Fecha_Comp_Indiv_Gar_6 = FALSE

            Ava_Cil_1_Gar_1 = TRUE
            Rec_Cil_1_Gar_1 = FALSE

            Ava_Cil_1_Gar_2 = TRUE
            Rec_Cil_1_Gar_2 = FALSE

            Ava_Cil_1_Gar_3 = TRUE
            Rec_Cil_1_Gar_3 = FALSE

            Ava_Cil_1_Gar_4 = TRUE
            Rec_Cil_1_Gar_4 = FALSE

            Ava_Cil_1_Gar_5 = TRUE
            Rec_Cil_1_Gar_5 = FALSE

            Ava_Cil_1_Gar_6 = TRUE
            Rec_Cil_1_Gar_6 = FALSE

            Ava_Cil_2_Gar_1 = TRUE
            Rec_Cil_2_Gar_1 = FALSE

            Ava_Cil_2_Gar_2 = TRUE
            Rec_Cil_2_Gar_2 = FALSE

            Ava_Cil_2_Gar_3 = TRUE
            Rec_Cil_2_Gar_3 = FALSE

            Ava_Cil_2_Gar_4 = TRUE
            Rec_Cil_2_Gar_4 = FALSE

            Ava_Cil_2_Gar_5 = TRUE
            Rec_Cil_2_Gar_5 = FALSE

            Ava_Cil_2_Gar_6 = TRUE
            Rec_Cil_2_Gar_6 = FALSE



         CASE 121
            Abre_Gar_Triplo_Lado_A = TRUE
            Fecha_Gar_Triplo_Lado_A = FALSE

            Abre_Gar_Triplo_Lado_B = TRUE
            Fecha_Gar_Triplo_Lado_B = FALSE

            Abre_Comp_Indiv_Gar_1 = FALSE
            Fecha_Comp_Indiv_Gar_1 = TRUE

            Abre_Comp_Indiv_Gar_3 = FALSE
            Fecha_Comp_Indiv_Gar_3 = TRUE

            Abre_Comp_Indiv_Gar_4 = FALSE
            Fecha_Comp_Indiv_Gar_4 = TRUE

            Abre_Comp_Indiv_Gar_6 = FALSE
            Fecha_Comp_Indiv_Gar_6 = TRUE

            Ava_Cil_1_Gar_1 = TRUE
            Rec_Cil_1_Gar_1 = FALSE

            Ava_Cil_1_Gar_2 = TRUE
            Rec_Cil_1_Gar_2 = FALSE

            Ava_Cil_1_Gar_3 = TRUE
            Rec_Cil_1_Gar_3 = FALSE

            Ava_Cil_1_Gar_4 = TRUE
            Rec_Cil_1_Gar_4 = FALSE

            Ava_Cil_1_Gar_5 = TRUE
            Rec_Cil_1_Gar_5 = FALSE

            Ava_Cil_1_Gar_6 = TRUE
            Rec_Cil_1_Gar_6 = FALSE

            Ava_Cil_2_Gar_1 = TRUE
            Rec_Cil_2_Gar_1 = FALSE

            Ava_Cil_2_Gar_2 = TRUE
            Rec_Cil_2_Gar_2 = FALSE

            Ava_Cil_2_Gar_3 = TRUE
            Rec_Cil_2_Gar_3 = FALSE

            Ava_Cil_2_Gar_4 = TRUE
            Rec_Cil_2_Gar_4 = FALSE

            Ava_Cil_2_Gar_5 = TRUE
            Rec_Cil_2_Gar_5 = FALSE

            Ava_Cil_2_Gar_6 = TRUE
            Rec_Cil_2_Gar_6 = FALSE



         CASE 122
            Abre_Gar_Triplo_Lado_A = TRUE
            Fecha_Gar_Triplo_Lado_A = FALSE

            Abre_Gar_Triplo_Lado_B = TRUE
            Fecha_Gar_Triplo_Lado_B = FALSE

            Abre_Comp_Indiv_Gar_1 = TRUE
            Fecha_Comp_Indiv_Gar_1 = FALSE

            Abre_Comp_Indiv_Gar_3 = FALSE
            Fecha_Comp_Indiv_Gar_3 = TRUE

            Abre_Comp_Indiv_Gar_4 = FALSE
            Fecha_Comp_Indiv_Gar_4 = TRUE

            Abre_Comp_Indiv_Gar_6 = TRUE
            Fecha_Comp_Indiv_Gar_6 = FALSE

            Ava_Cil_1_Gar_1 = TRUE
            Rec_Cil_1_Gar_1 = FALSE

            Ava_Cil_1_Gar_2 = TRUE
            Rec_Cil_1_Gar_2 = FALSE

            Ava_Cil_1_Gar_3 = TRUE
            Rec_Cil_1_Gar_3 = FALSE

            Ava_Cil_1_Gar_4 = TRUE
            Rec_Cil_1_Gar_4 = FALSE

            Ava_Cil_1_Gar_5 = TRUE
            Rec_Cil_1_Gar_5 = FALSE

            Ava_Cil_1_Gar_6 = TRUE
            Rec_Cil_1_Gar_6 = FALSE

            Ava_Cil_2_Gar_1 = TRUE
            Rec_Cil_2_Gar_1 = FALSE

            Ava_Cil_2_Gar_2 = TRUE
            Rec_Cil_2_Gar_2 = FALSE

            Ava_Cil_2_Gar_3 = TRUE
            Rec_Cil_2_Gar_3 = FALSE

            Ava_Cil_2_Gar_4 = TRUE
            Rec_Cil_2_Gar_4 = FALSE

            Ava_Cil_2_Gar_5 = TRUE
            Rec_Cil_2_Gar_5 = FALSE

            Ava_Cil_2_Gar_6 = TRUE
            Rec_Cil_2_Gar_6 = FALSE



         CASE 31
            Abre_Gar_Triplo_Lado_A = TRUE
            Fecha_Gar_Triplo_Lado_A = FALSE

            Abre_Gar_Triplo_Lado_B = TRUE
            Fecha_Gar_Triplo_Lado_B = FALSE

            Abre_Comp_Indiv_Gar_1 = FALSE
            Fecha_Comp_Indiv_Gar_1 = TRUE

            Abre_Comp_Indiv_Gar_3 = FALSE
            Fecha_Comp_Indiv_Gar_3 = TRUE

            Abre_Comp_Indiv_Gar_4 = FALSE
            Fecha_Comp_Indiv_Gar_4 = TRUE

            Abre_Comp_Indiv_Gar_6 = FALSE
            Fecha_Comp_Indiv_Gar_6 = TRUE

            Ava_Cil_1_Gar_1 = TRUE
            Rec_Cil_1_Gar_1 = FALSE

            Ava_Cil_1_Gar_2 = TRUE
            Rec_Cil_1_Gar_2 = FALSE

            Ava_Cil_1_Gar_3 = TRUE
            Rec_Cil_1_Gar_3 = FALSE

            Ava_Cil_1_Gar_4 = TRUE
            Rec_Cil_1_Gar_4 = FALSE

            Ava_Cil_1_Gar_5 = TRUE
            Rec_Cil_1_Gar_5 = FALSE

            Ava_Cil_1_Gar_6 = TRUE
            Rec_Cil_1_Gar_6 = FALSE

            Ava_Cil_2_Gar_1 = TRUE
            Rec_Cil_2_Gar_1 = FALSE

            Ava_Cil_2_Gar_2 = TRUE
            Rec_Cil_2_Gar_2 = FALSE

            Ava_Cil_2_Gar_3 = TRUE
            Rec_Cil_2_Gar_3 = FALSE

            Ava_Cil_2_Gar_4 = TRUE
            Rec_Cil_2_Gar_4 = FALSE

            Ava_Cil_2_Gar_5 = TRUE
            Rec_Cil_2_Gar_5 = FALSE

            Ava_Cil_2_Gar_6 = TRUE
            Rec_Cil_2_Gar_6 = FALSE


         CASE 32
            Abre_Gar_Triplo_Lado_A = TRUE
            Fecha_Gar_Triplo_Lado_A = FALSE

            Abre_Gar_Triplo_Lado_B = TRUE
            Fecha_Gar_Triplo_Lado_B = FALSE

            Abre_Comp_Indiv_Gar_1 = FALSE
            Fecha_Comp_Indiv_Gar_1 = TRUE

            Abre_Comp_Indiv_Gar_3 = FALSE
            Fecha_Comp_Indiv_Gar_3 = TRUE

            Abre_Comp_Indiv_Gar_4 = FALSE
            Fecha_Comp_Indiv_Gar_4 = TRUE

            Abre_Comp_Indiv_Gar_6 = FALSE
            Fecha_Comp_Indiv_Gar_6 = TRUE

            Ava_Cil_1_Gar_1 = TRUE
            Rec_Cil_1_Gar_1 = FALSE

            Ava_Cil_1_Gar_2 = TRUE
            Rec_Cil_1_Gar_2 = FALSE

            Ava_Cil_1_Gar_3 = TRUE
            Rec_Cil_1_Gar_3 = FALSE

            Ava_Cil_1_Gar_4 = TRUE
            Rec_Cil_1_Gar_4 = FALSE

            Ava_Cil_1_Gar_5 = TRUE
            Rec_Cil_1_Gar_5 = FALSE

            Ava_Cil_1_Gar_6 = TRUE
            Rec_Cil_1_Gar_6 = FALSE

            Ava_Cil_2_Gar_1 = TRUE
            Rec_Cil_2_Gar_1 = FALSE

            Ava_Cil_2_Gar_2 = TRUE
            Rec_Cil_2_Gar_2 = FALSE

            Ava_Cil_2_Gar_3 = TRUE
            Rec_Cil_2_Gar_3 = FALSE

            Ava_Cil_2_Gar_4 = TRUE
            Rec_Cil_2_Gar_4 = FALSE

            Ava_Cil_2_Gar_5 = TRUE
            Rec_Cil_2_Gar_5 = FALSE

            Ava_Cil_2_Gar_6 = TRUE
            Rec_Cil_2_Gar_6 = FALSE



         CASE 111
            Abre_Gar_Triplo_Lado_A = TRUE
            Fecha_Gar_Triplo_Lado_A = FALSE

            Abre_Gar_Triplo_Lado_B = TRUE
            Fecha_Gar_Triplo_Lado_B = FALSE

            Abre_Comp_Indiv_Gar_1 = FALSE
            Fecha_Comp_Indiv_Gar_1 = TRUE

            Abre_Comp_Indiv_Gar_3 = FALSE
            Fecha_Comp_Indiv_Gar_3 = TRUE

            Abre_Comp_Indiv_Gar_4 = FALSE
            Fecha_Comp_Indiv_Gar_4 = TRUE

            Abre_Comp_Indiv_Gar_6 = FALSE
            Fecha_Comp_Indiv_Gar_6 = TRUE

            Ava_Cil_1_Gar_1 = TRUE
            Rec_Cil_1_Gar_1 = FALSE

            Ava_Cil_1_Gar_2 = TRUE
            Rec_Cil_1_Gar_2 = FALSE

            Ava_Cil_1_Gar_3 = TRUE
            Rec_Cil_1_Gar_3 = FALSE

            Ava_Cil_1_Gar_4 = TRUE
            Rec_Cil_1_Gar_4 = FALSE

            Ava_Cil_1_Gar_5 = TRUE
            Rec_Cil_1_Gar_5 = FALSE

            Ava_Cil_1_Gar_6 = TRUE
            Rec_Cil_1_Gar_6 = FALSE

            Ava_Cil_2_Gar_1 = TRUE
            Rec_Cil_2_Gar_1 = FALSE

            Ava_Cil_2_Gar_2 = TRUE
            Rec_Cil_2_Gar_2 = FALSE

            Ava_Cil_2_Gar_3 = TRUE
            Rec_Cil_2_Gar_3 = FALSE

            Ava_Cil_2_Gar_4 = TRUE
            Rec_Cil_2_Gar_4 = FALSE

            Ava_Cil_2_Gar_5 = TRUE
            Rec_Cil_2_Gar_5 = FALSE

            Ava_Cil_2_Gar_6 = TRUE
            Rec_Cil_2_Gar_6 = FALSE



         CASE 112
            Abre_Gar_Triplo_Lado_A = TRUE
            Fecha_Gar_Triplo_Lado_A = FALSE

            Abre_Gar_Triplo_Lado_B = TRUE
            Fecha_Gar_Triplo_Lado_B = FALSE

            Abre_Comp_Indiv_Gar_1 = FALSE
            Fecha_Comp_Indiv_Gar_1 = TRUE

            Abre_Comp_Indiv_Gar_3 = FALSE
            Fecha_Comp_Indiv_Gar_3 = TRUE

            Abre_Comp_Indiv_Gar_4 = FALSE
            Fecha_Comp_Indiv_Gar_4 = TRUE

            Abre_Comp_Indiv_Gar_6 = FALSE
            Fecha_Comp_Indiv_Gar_6 = TRUE

            Ava_Cil_1_Gar_1 = TRUE
            Rec_Cil_1_Gar_1 = FALSE

            Ava_Cil_1_Gar_2 = TRUE
            Rec_Cil_1_Gar_2 = FALSE

            Ava_Cil_1_Gar_3 = TRUE
            Rec_Cil_1_Gar_3 = FALSE

            Ava_Cil_1_Gar_4 = TRUE
            Rec_Cil_1_Gar_4 = FALSE

            Ava_Cil_1_Gar_5 = TRUE
            Rec_Cil_1_Gar_5 = FALSE

            Ava_Cil_1_Gar_6 = TRUE
            Rec_Cil_1_Gar_6 = FALSE

            Ava_Cil_2_Gar_1 = TRUE
            Rec_Cil_2_Gar_1 = FALSE

            Ava_Cil_2_Gar_2 = TRUE
            Rec_Cil_2_Gar_2 = FALSE

            Ava_Cil_2_Gar_3 = TRUE
            Rec_Cil_2_Gar_3 = FALSE

            Ava_Cil_2_Gar_4 = TRUE
            Rec_Cil_2_Gar_4 = FALSE

            Ava_Cil_2_Gar_5 = TRUE
            Rec_Cil_2_Gar_5 = FALSE

            Ava_Cil_2_Gar_6 = TRUE
            Rec_Cil_2_Gar_6 = FALSE


         CASE 161
            Abre_Gar_Triplo_Lado_A = TRUE
            Fecha_Gar_Triplo_Lado_A = FALSE

            Abre_Gar_Triplo_Lado_B = TRUE
            Fecha_Gar_Triplo_Lado_B = FALSE

